LIN {X 0,Y 108.174,Z 556.008,A -85,B 0,C 180,E1 -26292.962,E2 -26292.962} C_VEL
LIN {X 0,Y 107.903,Z 556.034,A -85,B 0,C 180,E1 -26299.008,E2 -26299.008} C_VEL
LIN {X 0,Y 107.859,Z 556.038,A -85,B 0,C 180,E1 -26304.247,E2 -26304.247} C_VEL
LIN {X 0,Y 108.791,Z 558.837,A -85,B 0,C 180,E1 -26305.228,E2 -26305.228} C_VEL
LIN {X 0,Y 110.959,Z 561.09,A -85,B 0,C 180,E1 -26306.828,E2 -26306.828} C_VEL
LIN {X 0,Y 113.315,Z 564.846,A -85,B 0,C 180,E1 -26308.604,E2 -26308.604} C_VEL
LIN {X 0,Y 114.759,Z 566.953,A -85,B 0,C 180,E1 -26309.608,E2 -26309.608} C_VEL
LIN {X 0,Y 119.458,Z 573.968,A -85,B 0,C 180,E1 -26312.627,E2 -26312.627} C_VEL
LIN {X 0,Y 123.093,Z 581.209,A -85,B 0,C 180,E1 -26314.912,E2 -26314.912} C_VEL
LIN {X 0,Y 127.55,Z 591.655,A -85,B 0,C 180,E1 -26317.589,E2 -26317.589} C_VEL
LIN {X 0,Y 132.802,Z 606.179,A -85,B 0,C 180,E1 -26320.632,E2 -26320.632} C_VEL
LIN {X 0,Y 135.067,Z 613.749,A -85,B 0,C 180,E1 -26321.938,E2 -26321.938} C_VEL
LIN {X 0,Y 135.827,Z 626.997,A -85,B 0,C 180,E1 -26323.168,E2 -26323.168} C_VEL
LIN {X 0,Y 132.836,Z 662.155,A -85,B 0,C 180,E1 -26325.068,E2 -26325.068} C_VEL
LIN {X 0,Y 130.992,Z 674.498,A -85,B 0,C 180,E1 -26326.177,E2 -26326.177} C_VEL
LIN {X 0,Y 128.248,Z 687.244,A -85,B 0,C 180,E1 -26327.834,E2 -26327.834} C_VEL
LIN {X 0,Y 124.808,Z 699.792,A -85,B 0,C 180,E1 -26330.17,E2 -26330.17} C_VEL
LIN {X 0,Y 121.198,Z 711.054,A -85,B 0,C 180,E1 -26333.015,E2 -26333.015} C_VEL
LIN {X 0,Y 117.501,Z 721.244,A -85,B 0,C 180,E1 -26336.41,E2 -26336.41} C_VEL
LIN {X 0,Y 113.958,Z 730.437,A -85,B 0,C 180,E1 -26340.438,E2 -26340.438} C_VEL
LIN {X 0,Y 110.529,Z 739.404,A -85,B 0,C 180,E1 -26345.588,E2 -26345.588} C_VEL
LIN {X 0,Y 107.952,Z 746.556,A -85,B 0,C 180,E1 -26351.004,E2 -26351.004} C_VEL
LIN {X 0,Y 106.36,Z 752.228,A -85,B 0,C 180,E1 -26356.628,E2 -26356.628} C_VEL
LIN {X 0,Y 105.688,Z 756.645,A -85,B 0,C 180,E1 -26362.357,E2 -26362.357} C_VEL
LIN {X 0,Y 105.699,Z 758.945,A -85,B 0,C 180,E1 -26366.188,E2 -26366.188} C_VEL
LIN {X 0,Y 105.856,Z 760.773,A -85,B 0,C 180,E1 -26370,E2 -26370} C_VEL
LIN {X 0,Y 105.561,Z 762.058,A -85,B 0,C 180,E1 -26373.817,E2 -26373.817} C_VEL
LIN {X 0,Y 105.804,Z 763.39,A -85,B 0,C 180,E1 -26381.494,E2 -26381.494} C_VEL
LIN {X 0,Y 107.796,Z 763.255,A -85,B 0,C 180,E1 -26389.025,E2 -26389.025} C_VEL
LIN {X 0,Y 111.779,Z 761.601,A -85,B 0,C 180,E1 -26396.111,E2 -26396.111} C_VEL
LIN {X 0,Y 117.427,Z 758.445,A -85,B 0,C 180,E1 -26402.591,E2 -26402.591} C_VEL
LIN {X 0,Y 122.535,Z 755.011,A -85,B 0,C 180,E1 -26407.029,E2 -26407.029} C_VEL
LIN {X 0,Y 128.434,Z 750.585,A -85,B 0,C 180,E1 -26411.043,E2 -26411.043} C_VEL
LIN {X 0,Y 136.128,Z 744.032,A -85,B 0,C 180,E1 -26415.224,E2 -26415.224} C_VEL
LIN {X 0,Y 143.408,Z 736.982,A -85,B 0,C 180,E1 -26418.36,E2 -26418.36} C_VEL
LIN {X 0,Y 151.083,Z 728.338,A -85,B 0,C 180,E1 -26421.183,E2 -26421.183} C_VEL
LIN {X 0,Y 157.807,Z 719.589,A -85,B 0,C 180,E1 -26423.285,E2 -26423.285} C_VEL
LIN {X 0,Y 164.827,Z 708.925,A -85,B 0,C 180,E1 -26425.162,E2 -26425.162} C_VEL
LIN {X 0,Y 166.611,Z 705.818,A -85,B 0,C 180,E1 -26425.606,E2 -26425.606} C_VEL
LIN {X 0,Y 169.05,Z 701.001,A -85,B 0,C 180,E1 -26426.427,E2 -26426.427} C_VEL
LIN {X 0,Y 172.027,Z 693.095,A -85,B 0,C 180,E1 -26428.171,E2 -26428.171} C_VEL
LIN {X 0,Y 174.685,Z 684.872,A -85,B 0,C 180,E1 -26429.755,E2 -26429.755} C_VEL
LIN {X 0,Y 176.474,Z 679.565,A -85,B 0,C 180,E1 -26430.348,E2 -26430.348} C_VEL
LIN {X 0,Y 180.32,Z 666.962,A -85,B 0,C 180,E1 -26431.026,E2 -26431.026} C_VEL
LIN {X 0,Y 183.006,Z 653.633,A -85,B 0,C 180,E1 -26431.546,E2 -26431.546} C_VEL
LIN {X 0,Y 183.302,Z 651.418,A -85,B 0,C 180,E1 -26431.674,E2 -26431.674} C_VEL
LIN {X 0,Y 182.371,Z 646.522,A -85,B 0,C 180,E1 -26434.497,E2 -26434.497} C_VEL
LIN {X 0,Y 181.708,Z 643.146,A -85,B 0,C 180,E1 -26437.408,E2 -26437.408} C_VEL
LIN {X 0,Y 181.435,Z 641.338,A -85,B 0,C 180,E1 -26440.719,E2 -26440.719} C_VEL
LIN {X 0,Y 181.844,Z 641.486,A -85,B 0,C 180,E1 -26445.058,E2 -26445.058} C_VEL
LIN {X 0,Y 182.153,Z 642.109,A -85,B 0,C 180,E1 -26446.471,E2 -26446.471} C_VEL
LIN {X 0,Y 183.563,Z 645.549,A -85,B 0,C 180,E1 -26450.36,E2 -26450.36} C_VEL
LIN {X 0,Y 183.824,Z 646.592,A -85,B 0,C 180,E1 -26451.003,E2 -26451.003} C_VEL
LIN {X 0,Y 181.304,Z 660.599,A -85,B 0,C 180,E1 -26451.676,E2 -26451.676} C_VEL
LIN {X 0,Y 177.981,Z 672.516,A -85,B 0,C 180,E1 -26452.421,E2 -26452.421} C_VEL
LIN {X 0,Y 173.515,Z 684.485,A -85,B 0,C 180,E1 -26453.506,E2 -26453.506} C_VEL
LIN {X 0,Y 167.67,Z 696.546,A -85,B 0,C 180,E1 -26454.962,E2 -26454.962} C_VEL
LIN {X 0,Y 160.872,Z 707.775,A -85,B 0,C 180,E1 -26456.766,E2 -26456.766} C_VEL
LIN {X 0,Y 153.414,Z 717.859,A -85,B 0,C 180,E1 -26459.021,E2 -26459.021} C_VEL
LIN {X 0,Y 146.181,Z 726.118,A -85,B 0,C 180,E1 -26461.47,E2 -26461.47} C_VEL
LIN {X 0,Y 139.25,Z 732.906,A -85,B 0,C 180,E1 -26464.196,E2 -26464.196} C_VEL
LIN {X 0,Y 131.246,Z 739.533,A -85,B 0,C 180,E1 -26467.855,E2 -26467.855} C_VEL
LIN {X 0,Y 125.299,Z 743.757,A -85,B 0,C 180,E1 -26471.127,E2 -26471.127} C_VEL
LIN {X 0,Y 119.48,Z 747.278,A -85,B 0,C 180,E1 -26474.923,E2 -26474.923} C_VEL
LIN {X 0,Y 112.607,Z 750.675,A -85,B 0,C 180,E1 -26480.585,E2 -26480.585} C_VEL
LIN {X 0,Y 106.482,Z 752.713,A -85,B 0,C 180,E1 -26487.515,E2 -26487.515} C_VEL
LIN {X 0,Y 102.231,Z 753.183,A -85,B 0,C 180,E1 -26494.418,E2 -26494.418} C_VEL
LIN {X 0,Y 100.171,Z 752.678,A -85,B 0,C 180,E1 -26499.489,E2 -26499.489} C_VEL
LIN {X 0,Y 98.606,Z 751.336,A -85,B 0,C 180,E1 -26505.455,E2 -26505.455} C_VEL
LIN {X 0,Y 97.956,Z 748.857,A -85,B 0,C 180,E1 -26512.109,E2 -26512.109} C_VEL
LIN {X 0,Y 98.45,Z 745.149,A -85,B 0,C 180,E1 -26518.937,E2 -26518.937} C_VEL
LIN {X 0,Y 100.058,Z 739.9,A -85,B 0,C 180,E1 -26525.934,E2 -26525.934} C_VEL
LIN {X 0,Y 102.102,Z 734.278,A -85,B 0,C 180,E1 -26531.582,E2 -26531.582} C_VEL
LIN {X 0,Y 105.198,Z 726.618,A -85,B 0,C 180,E1 -26537.46,E2 -26537.46} C_VEL
LIN {X 0,Y 108.794,Z 717.855,A -85,B 0,C 180,E1 -26542.577,E2 -26542.577} C_VEL
LIN {X 0,Y 112.615,Z 708.271,A -85,B 0,C 180,E1 -26546.849,E2 -26546.849} C_VEL
LIN {X 0,Y 116.423,Z 697.687,A -85,B 0,C 180,E1 -26550.419,E2 -26550.419} C_VEL
LIN {X 0,Y 120.088,Z 686.177,A -85,B 0,C 180,E1 -26553.355,E2 -26553.355} C_VEL
LIN {X 0,Y 123.278,Z 673.736,A -85,B 0,C 180,E1 -26555.726,E2 -26555.726} C_VEL
LIN {X 0,Y 125.95,Z 660.371,A -85,B 0,C 180,E1 -26557.516,E2 -26557.516} C_VEL
LIN {X 0,Y 127.681,Z 647.584,A -85,B 0,C 180,E1 -26558.677,E2 -26558.677} C_VEL
LIN {X 0,Y 130.987,Z 609.66,A -85,B 0,C 180,E1 -26560.71,E2 -26560.71} C_VEL
LIN {X 0,Y 126.196,Z 597.94,A -85,B 0,C 180,E1 -26563.382,E2 -26563.382} C_VEL
LIN {X 0,Y 118.263,Z 583.132,A -85,B 0,C 180,E1 -26568.048,E2 -26568.048} C_VEL
LIN {X 0,Y 111.781,Z 573.193,A -85,B 0,C 180,E1 -26572.338,E2 -26572.338} C_VEL
LIN {X 0,Y 109.745,Z 570.24,A -85,B 0,C 180,E1 -26573.837,E2 -26573.837} C_VEL
LIN {X 0,Y 107.325,Z 566.668,A -85,B 0,C 180,E1 -26575.766,E2 -26575.766} C_VEL
LIN {X 0,Y 104.957,Z 563.637,A -85,B 0,C 180,E1 -26577.736,E2 -26577.736} C_VEL
LIN {X 0,Y 104.04,Z 562.118,A -85,B 0,C 180,E1 -26578.583,E2 -26578.583} C_VEL
LIN {X 0,Y 101.846,Z 560.004,A -85,B 0,C 180,E1 -26580.508,E2 -26580.508} C_VEL
LIN {X 0,Y 100.884,Z 557.533,A -85,B 0,C 180,E1 -26581.636,E2 -26581.636} C_VEL
LIN {X 0,Y 100.774,Z 556.932,A -85,B 0,C 180,E1 -26581.93,E2 -26581.93} C_VEL
LIN {X 0,Y 100.73,Z 556.92,A -85,B 0,C 180,E1 -26589.875,E2 -26589.875} C_VEL
LIN {X 0,Y 100.746,Z 556.92,A -85,B 0,C 180,E1 -26595.769,E2 -26595.769} C_VEL
LIN {X 0,Y 100.726,Z 556.931,A -85,B 0,C 180,E1 -26601.103,E2 -26601.103} C_VEL
LIN {X 0,Y 100.706,Z 556.915,A -85,B 0,C 180,E1 -26606.869,E2 -26606.869} C_VEL
LIN {X 0,Y 100.783,Z 556.926,A -85,B 0,C 180,E1 -26615.268,E2 -26615.268} C_VEL
LIN {X 0,Y 100.812,Z 556.897,A -85,B 0,C 180,E1 -26619.602,E2 -26619.602} C_VEL
LIN {X 0,Y 101.184,Z 556.859,A -85,B 0,C 180,E1 -26627.975,E2 -26627.975} C_VEL
LIN {X 0,Y 101.263,Z 556.844,A -85,B 0,C 180,E1 -26632.023,E2 -26632.023} C_VEL
LIN {X 0,Y 101.867,Z 556.767,A -85,B 0,C 180,E1 -26640.002,E2 -26640.002} C_VEL
LIN {X 0,Y 101.245,Z 556.856,A -85,B 0,C 180,E1 -26647.982,E2 -26647.982} C_VEL
LIN {X 0,Y 101.103,Z 556.89,A -85,B 0,C 180,E1 -26653.304,E2 -26653.304} C_VEL
LIN {X 0,Y 100.862,Z 557.093,A -85,B 0,C 180,E1 -26659.33,E2 -26659.33} C_VEL
LIN {X 0,Y 101.695,Z 559.548,A -85,B 0,C 180,E1 -26660.349,E2 -26660.349} C_VEL
LIN {X 0,Y 103.691,Z 561.773,A -85,B 0,C 180,E1 -26662.151,E2 -26662.151} C_VEL
LIN {X 0,Y 104.434,Z 562.453,A -85,B 0,C 180,E1 -26662.767,E2 -26662.767} C_VEL
LIN {X 0,Y 106.317,Z 565.65,A -85,B 0,C 180,E1 -26664.46,E2 -26664.46} C_VEL
LIN {X 0,Y 107.94,Z 567.61,A -85,B 0,C 180,E1 -26665.756,E2 -26665.756} C_VEL
LIN {X 0,Y 113.394,Z 575.832,A -85,B 0,C 180,E1 -26669.827,E2 -26669.827} C_VEL
LIN {X 0,Y 116.738,Z 581.563,A -85,B 0,C 180,E1 -26672.094,E2 -26672.094} C_VEL
LIN {X 0,Y 122.043,Z 593.85,A -85,B 0,C 180,E1 -26675.636,E2 -26675.636} C_VEL
LIN {X 0,Y 127.478,Z 609.128,A -85,B 0,C 180,E1 -26679.046,E2 -26679.046} C_VEL
LIN {X 0,Y 129.395,Z 615.319,A -85,B 0,C 180,E1 -26680.23,E2 -26680.23} C_VEL
LIN {X 0,Y 129.944,Z 628.507,A -85,B 0,C 180,E1 -26681.481,E2 -26681.481} C_VEL
LIN {X 0,Y 126.942,Z 661.822,A -85,B 0,C 180,E1 -26683.326,E2 -26683.326} C_VEL
LIN {X 0,Y 124.843,Z 675.074,A -85,B 0,C 180,E1 -26684.564,E2 -26684.564} C_VEL
LIN {X 0,Y 122.013,Z 687.548,A -85,B 0,C 180,E1 -26686.276,E2 -26686.276} C_VEL
LIN {X 0,Y 118.426,Z 699.92,A -85,B 0,C 180,E1 -26688.685,E2 -26688.685} C_VEL
LIN {X 0,Y 114.667,Z 711.088,A -85,B 0,C 180,E1 -26691.644,E2 -26691.644} C_VEL
LIN {X 0,Y 110.828,Z 721.179,A -85,B 0,C 180,E1 -26695.2,E2 -26695.2} C_VEL
LIN {X 0,Y 107.103,Z 730.309,A -85,B 0,C 180,E1 -26699.434,E2 -26699.434} C_VEL
LIN {X 0,Y 103.543,Z 739.234,A -85,B 0,C 180,E1 -26704.899,E2 -26704.899} C_VEL
LIN {X 0,Y 100.866,Z 746.322,A -85,B 0,C 180,E1 -26710.673,E2 -26710.673} C_VEL
LIN {X 0,Y 99.063,Z 752.766,A -85,B 0,C 180,E1 -26717.712,E2 -26717.712} C_VEL
LIN {X 0,Y 98.604,Z 756.946,A -85,B 0,C 180,E1 -26723.863,E2 -26723.863} C_VEL
LIN {X 0,Y 98.792,Z 759.978,A -85,B 0,C 180,E1 -26730,E2 -26730} C_VEL
LIN {X 0,Y 98.48,Z 761.358,A -85,B 0,C 180,E1 -26734.092,E2 -26734.092} C_VEL
LIN {X 0,Y 98.424,Z 762.314,A -85,B 0,C 180,E1 -26738.21,E2 -26738.21} C_VEL
LIN {X 0,Y 99.706,Z 763.05,A -85,B 0,C 180,E1 -26746.376,E2 -26746.376} C_VEL
LIN {X 0,Y 103.03,Z 762.345,A -85,B 0,C 180,E1 -26754.159,E2 -26754.159} C_VEL
LIN {X 0,Y 105.416,Z 761.445,A -85,B 0,C 180,E1 -26757.819,E2 -26757.819} C_VEL
LIN {X 0,Y 111.485,Z 758.462,A -85,B 0,C 180,E1 -26764.565,E2 -26764.565} C_VEL
LIN {X 0,Y 118.928,Z 753.911,A -85,B 0,C 180,E1 -26770.544,E2 -26770.544} C_VEL
LIN {X 0,Y 125.415,Z 749.322,A -85,B 0,C 180,E1 -26774.464,E2 -26774.464} C_VEL
LIN {X 0,Y 133.776,Z 742.537,A -85,B 0,C 180,E1 -26778.47,E2 -26778.47} C_VEL
LIN {X 0,Y 142.731,Z 733.94,A -85,B 0,C 180,E1 -26781.981,E2 -26781.981} C_VEL
LIN {X 0,Y 150.93,Z 724.692,A -85,B 0,C 180,E1 -26784.574,E2 -26784.574} C_VEL
LIN {X 0,Y 158.746,Z 714.242,A -85,B 0,C 180,E1 -26786.68,E2 -26786.68} C_VEL
LIN {X 0,Y 165.375,Z 703.731,A -85,B 0,C 180,E1 -26788.204,E2 -26788.204} C_VEL
LIN {X 0,Y 171.418,Z 691.984,A -85,B 0,C 180,E1 -26789.425,E2 -26789.425} C_VEL
LIN {X 0,Y 176.474,Z 679.565,A -85,B 0,C 180,E1 -26790.348,E2 -26790.348} C_VEL
LIN {X 0,Y 177.566,Z 675.97,A -85,B 0,C 180,E1 -26790.789,E2 -26790.789} C_VEL
LIN {X 0,Y 179.512,Z 664.776,A -85,B 0,C 180,E1 -26793.131,E2 -26793.131} C_VEL
LIN {X 0,Y 180.209,Z 661.025,A -85,B 0,C 180,E1 -26793.496,E2 -26793.496} C_VEL
LIN {X 0,Y 181.288,Z 655.573,A -85,B 0,C 180,E1 -26793.701,E2 -26793.701} C_VEL
LIN {X 0,Y 180.849,Z 652.395,A -85,B 0,C 180,E1 -26795.779,E2 -26795.779} C_VEL
LIN {X 0,Y 180.526,Z 649.844,A -85,B 0,C 180,E1 -26798.12,E2 -26798.12} C_VEL
LIN {X 0,Y 180.385,Z 648.406,A -85,B 0,C 180,E1 -26800.602,E2 -26800.602} C_VEL
LIN {X 0,Y 180.635,Z 648.307,A -85,B 0,C 180,E1 -26804.195,E2 -26804.195} C_VEL
LIN {X 0,Y 180.93,Z 648.948,A -85,B 0,C 180,E1 -26805.948,E2 -26805.948} C_VEL
LIN {X 0,Y 181.783,Z 651.483,A -85,B 0,C 180,E1 -26808.985,E2 -26808.985} C_VEL
LIN {X 0,Y 178.929,Z 664.632,A -85,B 0,C 180,E1 -26809.663,E2 -26809.663} C_VEL
LIN {X 0,Y 175.422,Z 675.737,A -85,B 0,C 180,E1 -26810.391,E2 -26810.391} C_VEL
LIN {X 0,Y 170.55,Z 687.561,A -85,B 0,C 180,E1 -26811.481,E2 -26811.481} C_VEL
LIN {X 0,Y 164.386,Z 699.333,A -85,B 0,C 180,E1 -26812.918,E2 -26812.918} C_VEL
LIN {X 0,Y 157.501,Z 709.886,A -85,B 0,C 180,E1 -26814.627,E2 -26814.627} C_VEL
LIN {X 0,Y 149.558,Z 719.987,A -85,B 0,C 180,E1 -26816.888,E2 -26816.888} C_VEL
LIN {X 0,Y 142.328,Z 727.638,A -85,B 0,C 180,E1 -26819.191,E2 -26819.191} C_VEL
LIN {X 0,Y 133.649,Z 735.359,A -85,B 0,C 180,E1 -26822.428,E2 -26822.428} C_VEL
LIN {X 0,Y 124.692,Z 742.032,A -85,B 0,C 180,E1 -26826.471,E2 -26826.471} C_VEL
LIN {X 0,Y 117.771,Z 746.289,A -85,B 0,C 180,E1 -26830.311,E2 -26830.311} C_VEL
LIN {X 0,Y 109.665,Z 750.263,A -85,B 0,C 180,E1 -26836,E2 -26836} C_VEL
LIN {X 0,Y 104.893,Z 752.074,A -85,B 0,C 180,E1 -26840.282,E2 -26840.282} C_VEL
LIN {X 0,Y 100.767,Z 753.166,A -85,B 0,C 180,E1 -26844.952,E2 -26844.952} C_VEL
LIN {X 0,Y 96.946,Z 753.621,A -85,B 0,C 180,E1 -26850.492,E2 -26850.492} C_VEL
LIN {X 0,Y 93.915,Z 753.228,A -85,B 0,C 180,E1 -26856.772,E2 -26856.772} C_VEL
LIN {X 0,Y 91.867,Z 751.887,A -85,B 0,C 180,E1 -26863.51,E2 -26863.51} C_VEL
LIN {X 0,Y 90.882,Z 748.999,A -85,B 0,C 180,E1 -26871.784,E2 -26871.784} C_VEL
LIN {X 0,Y 91.592,Z 744.432,A -85,B 0,C 180,E1 -26880.37,E2 -26880.37} C_VEL
LIN {X 0,Y 93.465,Z 738.703,A -85,B 0,C 180,E1 -26887.916,E2 -26887.916} C_VEL
LIN {X 0,Y 95.974,Z 732.381,A -85,B 0,C 180,E1 -26894.178,E2 -26894.178} C_VEL
LIN {X 0,Y 99.392,Z 724.525,A -85,B 0,C 180,E1 -26900.101,E2 -26900.101} C_VEL
LIN {X 0,Y 103.613,Z 714.664,A -85,B 0,C 180,E1 -26905.624,E2 -26905.624} C_VEL
LIN {X 0,Y 107.806,Z 704.231,A -85,B 0,C 180,E1 -26910,E2 -26910} C_VEL
LIN {X 0,Y 111.982,Z 692.588,A -85,B 0,C 180,E1 -26913.598,E2 -26913.598} C_VEL
LIN {X 0,Y 115.588,Z 680.766,A -85,B 0,C 180,E1 -26916.327,E2 -26916.327} C_VEL
LIN {X 0,Y 118.473,Z 669.013,A -85,B 0,C 180,E1 -26918.314,E2 -26918.314} C_VEL
LIN {X 0,Y 120.883,Z 655.475,A -85,B 0,C 180,E1 -26919.939,E2 -26919.939} C_VEL
LIN {X 0,Y 122.474,Z 642.382,A -85,B 0,C 180,E1 -26920.909,E2 -26920.909} C_VEL
LIN {X 0,Y 125.157,Z 611.497,A -85,B 0,C 180,E1 -26922.599,E2 -26922.599} C_VEL
LIN {X 0,Y 121.457,Z 602.23,A -85,B 0,C 180,E1 -26924.84,E2 -26924.84} C_VEL
LIN {X 0,Y 114.318,Z 588.414,A -85,B 0,C 180,E1 -26929.398,E2 -26929.398} C_VEL
LIN {X 0,Y 108.146,Z 578.586,A -85,B 0,C 180,E1 -26933.816,E2 -26933.816} C_VEL
LIN {X 0,Y 103.85,Z 572.191,A -85,B 0,C 180,E1 -26937.391,E2 -26937.391} C_VEL
LIN {X 0,Y 101.308,Z 568.556,A -85,B 0,C 180,E1 -26939.715,E2 -26939.715} C_VEL
LIN {X 0,Y 98.51,Z 565.258,A -85,B 0,C 180,E1 -26942.472,E2 -26942.472} C_VEL
LIN {X 0,Y 97.581,Z 563.315,A -85,B 0,C 180,E1 -26943.605,E2 -26943.605} C_VEL
LIN {X 0,Y 95.114,Z 561.387,A -85,B 0,C 180,E1 -26946.289,E2 -26946.289} C_VEL
LIN {X 0,Y 93.877,Z 558.999,A -85,B 0,C 180,E1 -26948.013,E2 -26948.013} C_VEL
LIN {X 0,Y 93.661,Z 557.799,A -85,B 0,C 180,E1 -26948.667,E2 -26948.667} C_VEL
LIN {X 0,Y 93.646,Z 557.818,A -85,B 0,C 180,E1 -26952.487,E2 -26952.487} C_VEL
LIN {X 0,Y 93.643,Z 557.795,A -85,B 0,C 180,E1 -26958.633,E2 -26958.633} C_VEL
LIN {X 0,Y 93.62,Z 557.804,A -85,B 0,C 180,E1 -26965.664,E2 -26965.664} C_VEL
LIN {X 0,Y 93.666,Z 557.817,A -85,B 0,C 180,E1 -26974.207,E2 -26974.207} C_VEL
LIN {X 0,Y 93.688,Z 557.786,A -85,B 0,C 180,E1 -26977.973,E2 -26977.973} C_VEL
LIN {X 0,Y 94.088,Z 557.751,A -85,B 0,C 180,E1 -26987.053,E2 -26987.053} C_VEL
LIN {X 0,Y 94.196,Z 557.72,A -85,B 0,C 180,E1 -26991.42,E2 -26991.42} C_VEL
LIN {X 0,Y 94.793,Z 557.647,A -85,B 0,C 180,E1 -27000.002,E2 -27000.002} C_VEL
LIN {X 0,Y 94.177,Z 557.733,A -85,B 0,C 180,E1 -27008.586,E2 -27008.586} C_VEL
LIN {X 0,Y 94.077,Z 557.764,A -85,B 0,C 180,E1 -27012.953,E2 -27012.953} C_VEL
LIN {X 0,Y 94.789,Z 560.311,A -85,B 0,C 180,E1 -27014.208,E2 -27014.208} C_VEL
LIN {X 0,Y 96.581,Z 562.529,A -85,B 0,C 180,E1 -27016.387,E2 -27016.387} C_VEL
LIN {X 0,Y 97.783,Z 563.493,A -85,B 0,C 180,E1 -27017.653,E2 -27017.653} C_VEL
LIN {X 0,Y 99.624,Z 566.67,A -85,B 0,C 180,E1 -27019.714,E2 -27019.714} C_VEL
LIN {X 0,Y 101.343,Z 568.577,A -85,B 0,C 180,E1 -27021.339,E2 -27021.339} C_VEL
LIN {X 0,Y 103.777,Z 572.135,A -85,B 0,C 180,E1 -27023.564,E2 -27023.564} C_VEL
LIN {X 0,Y 109.381,Z 580.683,A -85,B 0,C 180,E1 -27028.157,E2 -27028.157} C_VEL
LIN {X 0,Y 112.465,Z 586.164,A -85,B 0,C 180,E1 -27030.434,E2 -27030.434} C_VEL
LIN {X 0,Y 117.395,Z 598.14,A -85,B 0,C 180,E1 -27034.047,E2 -27034.047} C_VEL
LIN {X 0,Y 122.249,Z 612.383,A -85,B 0,C 180,E1 -27037.391,E2 -27037.391} C_VEL
LIN {X 0,Y 123.866,Z 618.008,A -85,B 0,C 180,E1 -27038.49,E2 -27038.49} C_VEL
LIN {X 0,Y 124.205,Z 629.468,A -85,B 0,C 180,E1 -27039.601,E2 -27039.601} C_VEL
LIN {X 0,Y 121.204,Z 661.249,A -85,B 0,C 180,E1 -27041.395,E2 -27041.395} C_VEL
LIN {X 0,Y 119.119,Z 674.228,A -85,B 0,C 180,E1 -27042.639,E2 -27042.639} C_VEL
LIN {X 0,Y 116.147,Z 686.797,A -85,B 0,C 180,E1 -27044.377,E2 -27044.377} C_VEL
LIN {X 0,Y 112.659,Z 698.443,A -85,B 0,C 180,E1 -27046.67,E2 -27046.67} C_VEL
LIN {X 0,Y 108.7,Z 709.784,A -85,B 0,C 180,E1 -27049.719,E2 -27049.719} C_VEL
LIN {X 0,Y 105.062,Z 718.997,A -85,B 0,C 180,E1 -27052.985,E2 -27052.985} C_VEL
LIN {X 0,Y 101.042,Z 728.481,A -85,B 0,C 180,E1 -27057.382,E2 -27057.382} C_VEL
LIN {X 0,Y 97.114,Z 737.62,A -85,B 0,C 180,E1 -27063.109,E2 -27063.109} C_VEL
LIN {X 0,Y 94.187,Z 744.963,A -85,B 0,C 180,E1 -27069.242,E2 -27069.242} C_VEL
LIN {X 0,Y 92.548,Z 749.899,A -85,B 0,C 180,E1 -27074.587,E2 -27074.587} C_VEL
LIN {X 0,Y 91.622,Z 754.658,A -85,B 0,C 180,E1 -27081.175,E2 -27081.175} C_VEL
LIN {X 0,Y 91.588,Z 757.393,A -85,B 0,C 180,E1 -27086.024,E2 -27086.024} C_VEL
LIN {X 0,Y 91.73,Z 759.166,A -85,B 0,C 180,E1 -27090,E2 -27090} C_VEL
LIN {X 0,Y 91.411,Z 760.618,A -85,B 0,C 180,E1 -27094.409,E2 -27094.409} C_VEL
LIN {X 0,Y 91.9,Z 762.332,A -85,B 0,C 180,E1 -27103.263,E2 -27103.263} C_VEL
LIN {X 0,Y 94.422,Z 762.497,A -85,B 0,C 180,E1 -27111.848,E2 -27111.848} C_VEL
LIN {X 0,Y 99.161,Z 761.233,A -85,B 0,C 180,E1 -27119.743,E2 -27119.743} C_VEL
LIN {X 0,Y 105.693,Z 758.48,A -85,B 0,C 180,E1 -27126.758,E2 -27126.758} C_VEL
LIN {X 0,Y 113.615,Z 754.137,A -85,B 0,C 180,E1 -27132.876,E2 -27132.876} C_VEL
LIN {X 0,Y 120.47,Z 749.748,A -85,B 0,C 180,E1 -27136.82,E2 -27136.82} C_VEL
LIN {X 0,Y 129.201,Z 743.244,A -85,B 0,C 180,E1 -27140.816,E2 -27140.816} C_VEL
LIN {X 0,Y 138.515,Z 734.952,A -85,B 0,C 180,E1 -27144.271,E2 -27144.271} C_VEL
LIN {X 0,Y 146.99,Z 726.121,A -85,B 0,C 180,E1 -27146.793,E2 -27146.793} C_VEL
LIN {X 0,Y 155.052,Z 716.15,A -85,B 0,C 180,E1 -27148.817,E2 -27148.817} C_VEL
LIN {X 0,Y 162.581,Z 704.863,A -85,B 0,C 180,E1 -27150.451,E2 -27150.451} C_VEL
LIN {X 0,Y 168.768,Z 693.602,A -85,B 0,C 180,E1 -27151.604,E2 -27151.604} C_VEL
LIN {X 0,Y 174.518,Z 680.239,A -85,B 0,C 180,E1 -27152.562,E2 -27152.562} C_VEL
LIN {X 0,Y 178.785,Z 666.964,A -85,B 0,C 180,E1 -27153.238,E2 -27153.238} C_VEL
LIN {X 0,Y 180.209,Z 661.025,A -85,B 0,C 180,E1 -27153.496,E2 -27153.496} C_VEL
LIN {X 0,Y 180.487,Z 659.028,A -85,B 0,C 180,E1 -27153.833,E2 -27153.833} C_VEL
LIN {X 0,Y 180.462,Z 657.363,A -85,B 0,C 180,E1 -27154.636,E2 -27154.636} C_VEL
LIN {X 0,Y 180.075,Z 656.344,A -85,B 0,C 180,E1 -27156.041,E2 -27156.041} C_VEL
LIN {X 0,Y 179.126,Z 656.066,A -85,B 0,C 180,E1 -27159.577,E2 -27159.577} C_VEL
LIN {X 0,Y 179.108,Z 655.824,A -85,B 0,C 180,E1 -27160.078,E2 -27160.078} C_VEL
LIN {X 0,Y 179.118,Z 655.203,A -85,B 0,C 180,E1 -27161.705,E2 -27161.705} C_VEL
LIN {X 0,Y 179.507,Z 655.551,A -85,B 0,C 180,E1 -27165.248,E2 -27165.248} C_VEL
LIN {X 0,Y 179.709,Z 657.068,A -85,B 0,C 180,E1 -27167.008,E2 -27167.008} C_VEL
LIN {X 0,Y 176.409,Z 669.66,A -85,B 0,C 180,E1 -27167.655,E2 -27167.655} C_VEL
LIN {X 0,Y 171.611,Z 682.589,A -85,B 0,C 180,E1 -27168.606,E2 -27168.606} C_VEL
LIN {X 0,Y 166.028,Z 694.169,A -85,B 0,C 180,E1 -27169.779,E2 -27169.779} C_VEL
LIN {X 0,Y 159.079,Z 705.518,A -85,B 0,C 180,E1 -27171.298,E2 -27171.298} C_VEL
LIN {X 0,Y 152.252,Z 714.701,A -85,B 0,C 180,E1 -27172.941,E2 -27172.941} C_VEL
LIN {X 0,Y 144.482,Z 723.512,A -85,B 0,C 180,E1 -27175.043,E2 -27175.043} C_VEL
LIN {X 0,Y 135.679,Z 731.834,A -85,B 0,C 180,E1 -27177.779,E2 -27177.779} C_VEL
LIN {X 0,Y 126.528,Z 738.973,A -85,B 0,C 180,E1 -27181.189,E2 -27181.189} C_VEL
LIN {X 0,Y 119.787,Z 743.385,A -85,B 0,C 180,E1 -27184.15,E2 -27184.15} C_VEL
LIN {X 0,Y 110.388,Z 748.485,A -85,B 0,C 180,E1 -27189.318,E2 -27189.318} C_VEL
LIN {X 0,Y 102.041,Z 751.849,A -85,B 0,C 180,E1 -27195.374,E2 -27195.374} C_VEL
LIN {X 0,Y 95.78,Z 753.534,A -85,B 0,C 180,E1 -27201.521,E2 -27201.521} C_VEL
LIN {X 0,Y 91.209,Z 754.067,A -85,B 0,C 180,E1 -27207.534,E2 -27207.534} C_VEL
LIN {X 0,Y 86.898,Z 753.457,A -85,B 0,C 180,E1 -27216.027,E2 -27216.027} C_VEL
LIN {X 0,Y 85.054,Z 752.247,A -85,B 0,C 180,E1 -27221.957,E2 -27221.957} C_VEL
LIN {X 0,Y 83.805,Z 749.078,A -85,B 0,C 180,E1 -27231.492,E2 -27231.492} C_VEL
LIN {X 0,Y 84.38,Z 744.813,A -85,B 0,C 180,E1 -27240.018,E2 -27240.018} C_VEL
LIN {X 0,Y 86.434,Z 738.813,A -85,B 0,C 180,E1 -27248.538,E2 -27248.538} C_VEL
LIN {X 0,Y 88.866,Z 732.977,A -85,B 0,C 180,E1 -27254.759,E2 -27254.759} C_VEL
LIN {X 0,Y 92.543,Z 724.951,A -85,B 0,C 180,E1 -27261.264,E2 -27261.264} C_VEL
LIN {X 0,Y 96.545,Z 716.087,A -85,B 0,C 180,E1 -27266.605,E2 -27266.605} C_VEL
LIN {X 0,Y 101.195,Z 705.215,A -85,B 0,C 180,E1 -27271.492,E2 -27271.492} C_VEL
LIN {X 0,Y 105.07,Z 695.19,A -85,B 0,C 180,E1 -27274.838,E2 -27274.838} C_VEL
LIN {X 0,Y 109.058,Z 683.033,A -85,B 0,C 180,E1 -27277.871,E2 -27277.871} C_VEL
LIN {X 0,Y 112.344,Z 670.656,A -85,B 0,C 180,E1 -27280.133,E2 -27280.133} C_VEL
LIN {X 0,Y 114.861,Z 657.82,A -85,B 0,C 180,E1 -27281.775,E2 -27281.775} C_VEL
LIN {X 0,Y 116.717,Z 644.153,A -85,B 0,C 180,E1 -27282.87,E2 -27282.87} C_VEL
LIN {X 0,Y 119.53,Z 614.275,A -85,B 0,C 180,E1 -27284.515,E2 -27284.515} C_VEL
LIN {X 0,Y 119.018,Z 612.229,A -85,B 0,C 180,E1 -27284.916,E2 -27284.916} C_VEL
LIN {X 0,Y 116.634,Z 606.127,A -85,B 0,C 180,E1 -27286.53,E2 -27286.53} C_VEL
LIN {X 0,Y 109.897,Z 592.771,A -85,B 0,C 180,E1 -27291.199,E2 -27291.199} C_VEL
LIN {X 0,Y 103.336,Z 581.898,A -85,B 0,C 180,E1 -27296.487,E2 -27296.487} C_VEL
LIN {X 0,Y 99.931,Z 577.057,A -85,B 0,C 180,E1 -27299.569,E2 -27299.569} C_VEL
LIN {X 0,Y 97.593,Z 573.734,A -85,B 0,C 180,E1 -27301.957,E2 -27301.957} C_VEL
LIN {X 0,Y 95.178,Z 570.274,A -85,B 0,C 180,E1 -27304.714,E2 -27304.714} C_VEL
LIN {X 0,Y 94.58,Z 569.401,A -85,B 0,C 180,E1 -27305.444,E2 -27305.444} C_VEL
LIN {X 0,Y 92.116,Z 566.856,A -85,B 0,C 180,E1 -27308.481,E2 -27308.481} C_VEL
LIN {X 0,Y 90.825,Z 564.314,A -85,B 0,C 180,E1 -27310.506,E2 -27310.506} C_VEL
LIN {X 0,Y 88.01,Z 562.227,A -85,B 0,C 180,E1 -27314.851,E2 -27314.851} C_VEL
LIN {X 0,Y 86.896,Z 560.043,A -85,B 0,C 180,E1 -27317.216,E2 -27317.216} C_VEL
LIN {X 0,Y 86.602,Z 558.671,A -85,B 0,C 180,E1 -27318.16,E2 -27318.16} C_VEL
LIN {X 0,Y 86.57,Z 558.683,A -85,B 0,C 180,E1 -27325.373,E2 -27325.373} C_VEL
LIN {X 0,Y 86.581,Z 558.7,A -85,B 0,C 180,E1 -27333.237,E2 -27333.237} C_VEL
LIN {X 0,Y 86.642,Z 558.665,A -85,B 0,C 180,E1 -27341.07,E2 -27341.07} C_VEL
LIN {X 0,Y 86.967,Z 558.646,A -85,B 0,C 180,E1 -27345.972,E2 -27345.972} C_VEL
LIN {X 0,Y 87.104,Z 558.601,A -85,B 0,C 180,E1 -27350.716,E2 -27350.716} C_VEL
LIN {X 0,Y 87.721,Z 558.528,A -85,B 0,C 180,E1 -27360.002,E2 -27360.002} C_VEL
LIN {X 0,Y 87.271,Z 558.605,A -85,B 0,C 180,E1 -27364.043,E2 -27364.043} C_VEL
LIN {X 0,Y 87.865,Z 560.92,A -85,B 0,C 180,E1 -27365.597,E2 -27365.597} C_VEL
LIN {X 0,Y 89.645,Z 563.215,A -85,B 0,C 180,E1 -27368.739,E2 -27368.739} C_VEL
LIN {X 0,Y 91.398,Z 564.504,A -85,B 0,C 180,E1 -27371.226,E2 -27371.226} C_VEL
LIN {X 0,Y 93.01,Z 567.586,A -85,B 0,C 180,E1 -27373.621,E2 -27373.621} C_VEL
LIN {X 0,Y 95.062,Z 569.835,A -85,B 0,C 180,E1 -27376.141,E2 -27376.141} C_VEL
LIN {X 0,Y 97.508,Z 573.495,A -85,B 0,C 180,E1 -27378.962,E2 -27378.962} C_VEL
LIN {X 0,Y 98.888,Z 575.542,A -85,B 0,C 180,E1 -27380.409,E2 -27380.409} C_VEL
LIN {X 0,Y 101.918,Z 580.045,A -85,B 0,C 180,E1 -27383.304,E2 -27383.304} C_VEL
LIN {X 0,Y 105.825,Z 586.251,A -85,B 0,C 180,E1 -27386.695,E2 -27386.695} C_VEL
LIN {X 0,Y 108.188,Z 590.603,A -85,B 0,C 180,E1 -27388.611,E2 -27388.611} C_VEL
LIN {X 0,Y 112.866,Z 602.453,A -85,B 0,C 180,E1 -27392.344,E2 -27392.344} C_VEL
LIN {X 0,Y 117.303,Z 616.175,A -85,B 0,C 180,E1 -27395.745,E2 -27395.745} C_VEL
LIN {X 0,Y 118.368,Z 620.399,A -85,B 0,C 180,E1 -27396.586,E2 -27396.586} C_VEL
LIN {X 0,Y 118.642,Z 629.302,A -85,B 0,C 180,E1 -27397.518,E2 -27397.518} C_VEL
LIN {X 0,Y 115.562,Z 660.655,A -85,B 0,C 180,E1 -27399.332,E2 -27399.332} C_VEL
LIN {X 0,Y 113.378,Z 673.671,A -85,B 0,C 180,E1 -27400.595,E2 -27400.595} C_VEL
LIN {X 0,Y 110.146,Z 686.792,A -85,B 0,C 180,E1 -27402.461,E2 -27402.461} C_VEL
LIN {X 0,Y 106.511,Z 698.349,A -85,B 0,C 180,E1 -27404.821,E2 -27404.821} C_VEL
LIN {X 0,Y 102.371,Z 709.635,A -85,B 0,C 180,E1 -27407.983,E2 -27407.983} C_VEL
LIN {X 0,Y 98.45,Z 719.038,A -85,B 0,C 180,E1 -27411.49,E2 -27411.49} C_VEL
LIN {X 0,Y 94.32,Z 728.236,A -85,B 0,C 180,E1 -27416.025,E2 -27416.025} C_VEL
LIN {X 0,Y 90.205,Z 737.35,A -85,B 0,C 180,E1 -27422.131,E2 -27422.131} C_VEL
LIN {X 0,Y 87.121,Z 744.662,A -85,B 0,C 180,E1 -27428.715,E2 -27428.715} C_VEL
LIN {X 0,Y 85.196,Z 750.473,A -85,B 0,C 180,E1 -27435.672,E2 -27435.672} C_VEL
LIN {X 0,Y 84.484,Z 754.998,A -85,B 0,C 180,E1 -27442.832,E2 -27442.832} C_VEL
LIN {X 0,Y 84.67,Z 758.353,A -85,B 0,C 180,E1 -27450,E2 -27450} C_VEL
LIN {X 0,Y 84.345,Z 759.869,A -85,B 0,C 180,E1 -27454.78,E2 -27454.78} C_VEL
LIN {X 0,Y 85.001,Z 761.725,A -85,B 0,C 180,E1 -27464.361,E2 -27464.361} C_VEL
LIN {X 0,Y 87.841,Z 762.116,A -85,B 0,C 180,E1 -27473.58,E2 -27473.58} C_VEL
LIN {X 0,Y 93.035,Z 761.016,A -85,B 0,C 180,E1 -27481.923,E2 -27481.923} C_VEL
LIN {X 0,Y 100.079,Z 758.481,A -85,B 0,C 180,E1 -27489.198,E2 -27489.198} C_VEL
LIN {X 0,Y 106.274,Z 755.547,A -85,B 0,C 180,E1 -27493.976,E2 -27493.976} C_VEL
LIN {X 0,Y 113.253,Z 751.675,A -85,B 0,C 180,E1 -27498.129,E2 -27498.129} C_VEL
LIN {X 0,Y 120.843,Z 746.796,A -85,B 0,C 180,E1 -27501.731,E2 -27501.731} C_VEL
LIN {X 0,Y 130.356,Z 739.643,A -85,B 0,C 180,E1 -27505.303,E2 -27505.303} C_VEL
LIN {X 0,Y 138.878,Z 731.989,A -85,B 0,C 180,E1 -27507.954,E2 -27507.954} C_VEL
LIN {X 0,Y 147.764,Z 722.517,A -85,B 0,C 180,E1 -27510.226,E2 -27510.226} C_VEL
LIN {X 0,Y 156.166,Z 711.856,A -85,B 0,C 180,E1 -27512.027,E2 -27512.027} C_VEL
LIN {X 0,Y 163.205,Z 700.971,A -85,B 0,C 180,E1 -27513.319,E2 -27513.319} C_VEL
LIN {X 0,Y 169.587,Z 688.812,A -85,B 0,C 180,E1 -27514.335,E2 -27514.335} C_VEL
LIN {X 0,Y 174.205,Z 677.667,A -85,B 0,C 180,E1 -27515.001,E2 -27515.001} C_VEL
LIN {X 0,Y 178.265,Z 664.418,A -85,B 0,C 180,E1 -27515.607,E2 -27515.607} C_VEL
LIN {X 0,Y 179.314,Z 660.071,A -85,B 0,C 180,E1 -27515.756,E2 -27515.756} C_VEL
LIN {X 0,Y 179.185,Z 657.061,A -85,B 0,C 180,E1 -27518.1,E2 -27518.1} C_VEL
LIN {X 0,Y 179.108,Z 655.824,A -85,B 0,C 180,E1 -27520.078,E2 -27520.078} C_VEL
LIN {X 0,Y 179.02,Z 655.898,A -85,B 0,C 180,E1 -27521.19,E2 -27521.19} C_VEL
LIN {X 0,Y 178.715,Z 657.427,A -85,B 0,C 180,E1 -27522.457,E2 -27522.457} C_VEL
LIN {X 0,Y 178.096,Z 660.501,A -85,B 0,C 180,E1 -27523.738,E2 -27523.738} C_VEL
LIN {X 0,Y 177.334,Z 663.92,A -85,B 0,C 180,E1 -27524.632,E2 -27524.632} C_VEL
LIN {X 0,Y 176.267,Z 667.818,A -85,B 0,C 180,E1 -27525.217,E2 -27525.217} C_VEL
LIN {X 0,Y 175.856,Z 669.2,A -85,B 0,C 180,E1 -27525.324,E2 -27525.324} C_VEL
LIN {X 0,Y 171.401,Z 681.244,A -85,B 0,C 180,E1 -27526.119,E2 -27526.119} C_VEL
LIN {X 0,Y 165.789,Z 692.864,A -85,B 0,C 180,E1 -27527.155,E2 -27527.155} C_VEL
LIN {X 0,Y 159.438,Z 703.469,A -85,B 0,C 180,E1 -27528.408,E2 -27528.408} C_VEL
LIN {X 0,Y 152.663,Z 712.769,A -85,B 0,C 180,E1 -27529.822,E2 -27529.822} C_VEL
LIN {X 0,Y 144.082,Z 722.48,A -85,B 0,C 180,E1 -27531.875,E2 -27531.875} C_VEL
LIN {X 0,Y 135.977,Z 730.117,A -85,B 0,C 180,E1 -27534.065,E2 -27534.065} C_VEL
LIN {X 0,Y 126.668,Z 737.473,A -85,B 0,C 180,E1 -27537.055,E2 -27537.055} C_VEL
LIN {X 0,Y 118.939,Z 742.559,A -85,B 0,C 180,E1 -27539.998,E2 -27539.998} C_VEL
LIN {X 0,Y 111.006,Z 746.918,A -85,B 0,C 180,E1 -27543.628,E2 -27543.628} C_VEL
LIN {X 0,Y 103.612,Z 750.208,A -85,B 0,C 180,E1 -27547.795,E2 -27547.795} C_VEL
LIN {X 0,Y 96.856,Z 752.529,A -85,B 0,C 180,E1 -27552.571,E2 -27552.571} C_VEL
LIN {X 0,Y 89.482,Z 754.206,A -85,B 0,C 180,E1 -27559.53,E2 -27559.53} C_VEL
LIN {X 0,Y 85.243,Z 754.52,A -85,B 0,C 180,E1 -27564.921,E2 -27564.921} C_VEL
LIN {X 0,Y 81.683,Z 754.196,A -85,B 0,C 180,E1 -27571.077,E2 -27571.077} C_VEL
LIN {X 0,Y 78.688,Z 752.949,A -85,B 0,C 180,E1 -27578.694,E2 -27578.694} C_VEL
LIN {X 0,Y 77.023,Z 750.694,A -85,B 0,C 180,E1 -27586.88,E2 -27586.88} C_VEL
LIN {X 0,Y 76.892,Z 746.636,A -85,B 0,C 180,E1 -27596.743,E2 -27596.743} C_VEL
LIN {X 0,Y 78.037,Z 742.424,A -85,B 0,C 180,E1 -27604.231,E2 -27604.231} C_VEL
LIN {X 0,Y 80.126,Z 737.165,A -85,B 0,C 180,E1 -27611.39,E2 -27611.39} C_VEL
LIN {X 0,Y 83.583,Z 729.638,A -85,B 0,C 180,E1 -27619.095,E2 -27619.095} C_VEL
LIN {X 0,Y 87.628,Z 721.28,A -85,B 0,C 180,E1 -27625.4,E2 -27625.4} C_VEL
LIN {X 0,Y 92.012,Z 712.053,A -85,B 0,C 180,E1 -27630.547,E2 -27630.547} C_VEL
LIN {X 0,Y 96.652,Z 701.36,A -85,B 0,C 180,E1 -27634.998,E2 -27634.998} C_VEL
LIN {X 0,Y 101.047,Z 689.818,A -85,B 0,C 180,E1 -27638.499,E2 -27638.499} C_VEL
LIN {X 0,Y 105.095,Z 676.943,A -85,B 0,C 180,E1 -27641.328,E2 -27641.328} C_VEL
LIN {X 0,Y 108.184,Z 664.23,A -85,B 0,C 180,E1 -27643.295,E2 -27643.295} C_VEL
LIN {X 0,Y 110.5,Z 650.388,A -85,B 0,C 180,E1 -27644.738,E2 -27644.738} C_VEL
LIN {X 0,Y 114.014,Z 615.508,A -85,B 0,C 180,E1 -27646.794,E2 -27646.794} C_VEL
LIN {X 0,Y 111.943,Z 610.191,A -85,B 0,C 180,E1 -27648.295,E2 -27648.295} C_VEL
LIN {X 0,Y 105.791,Z 597.449,A -85,B 0,C 180,E1 -27652.991,E2 -27652.991} C_VEL
LIN {X 0,Y 99.63,Z 587.006,A -85,B 0,C 180,E1 -27658.403,E2 -27658.403} C_VEL
LIN {X 0,Y 94.931,Z 579.885,A -85,B 0,C 180,E1 -27663.359,E2 -27663.359} C_VEL
LIN {X 0,Y 92.363,Z 576.135,A -85,B 0,C 180,E1 -27666.504,E2 -27666.504} C_VEL
LIN {X 0,Y 89.398,Z 572.52,A -85,B 0,C 180,E1 -27670.585,E2 -27670.585} C_VEL
LIN {X 0,Y 88.452,Z 570.75,A -85,B 0,C 180,E1 -27672.216,E2 -27672.216} C_VEL
LIN {X 0,Y 86.014,Z 568.593,A -85,B 0,C 180,E1 -27676.416,E2 -27676.416} C_VEL
LIN {X 0,Y 84.688,Z 565.79,A -85,B 0,C 180,E1 -27679.587,E2 -27679.587} C_VEL
LIN {X 0,Y 84.004,Z 565.334,A -85,B 0,C 180,E1 -27681.14,E2 -27681.14} C_VEL
LIN {X 0,Y 80.349,Z 562.115,A -85,B 0,C 180,E1 -27696.823,E2 -27696.823} C_VEL
LIN {X 0,Y 80.605,Z 561.809,A -85,B 0,C 180,E1 -27706.313,E2 -27706.313} C_VEL
LIN {X 0,Y 85.15,Z 565.301,A -85,B 0,C 180,E1 -27722.131,E2 -27722.131} C_VEL
LIN {X 0,Y 86.386,Z 568.248,A -85,B 0,C 180,E1 -27725.107,E2 -27725.107} C_VEL
LIN {X 0,Y 89.053,Z 571.015,A -85,B 0,C 180,E1 -27729.657,E2 -27729.657} C_VEL
LIN {X 0,Y 91.009,Z 574.334,A -85,B 0,C 180,E1 -27732.688,E2 -27732.688} C_VEL
LIN {X 0,Y 92.466,Z 576.093,A -85,B 0,C 180,E1 -27734.585,E2 -27734.585} C_VEL
LIN {X 0,Y 95.821,Z 581.277,A -85,B 0,C 180,E1 -27738.701,E2 -27738.701} C_VEL
LIN {X 0,Y 99.795,Z 587.428,A -85,B 0,C 180,E1 -27742.771,E2 -27742.771} C_VEL
LIN {X 0,Y 103.962,Z 594.937,A -85,B 0,C 180,E1 -27746.591,E2 -27746.591} C_VEL
LIN {X 0,Y 108.158,Z 606.108,A -85,B 0,C 180,E1 -27750.345,E2 -27750.345} C_VEL
LIN {X 0,Y 112.541,Z 620.27,A -85,B 0,C 180,E1 -27754.029,E2 -27754.029} C_VEL
LIN {X 0,Y 113.064,Z 622.764,A -85,B 0,C 180,E1 -27754.524,E2 -27754.524} C_VEL
LIN {X 0,Y 113.089,Z 630.842,A -85,B 0,C 180,E1 -27755.345,E2 -27755.345} C_VEL
LIN {X 0,Y 109.934,Z 660.976,A -85,B 0,C 180,E1 -27757.13,E2 -27757.13} C_VEL
LIN {X 0,Y 107.643,Z 673.831,A -85,B 0,C 180,E1 -27758.421,E2 -27758.421} C_VEL
LIN {X 0,Y 104.552,Z 685.747,A -85,B 0,C 180,E1 -27760.128,E2 -27760.128} C_VEL
LIN {X 0,Y 100.494,Z 698.26,A -85,B 0,C 180,E1 -27762.752,E2 -27762.752} C_VEL
LIN {X 0,Y 96.148,Z 709.487,A -85,B 0,C 180,E1 -27766.021,E2 -27766.021} C_VEL
LIN {X 0,Y 91.654,Z 719.689,A -85,B 0,C 180,E1 -27770.07,E2 -27770.07} C_VEL
LIN {X 0,Y 86.876,Z 729.632,A -85,B 0,C 180,E1 -27775.51,E2 -27775.51} C_VEL
LIN {X 0,Y 82.724,Z 738.42,A -85,B 0,C 180,E1 -27782.144,E2 -27782.144} C_VEL
LIN {X 0,Y 79.701,Z 745.385,A -85,B 0,C 180,E1 -27789.347,E2 -27789.347} C_VEL
LIN {X 0,Y 77.9,Z 750.92,A -85,B 0,C 180,E1 -27796.965,E2 -27796.965} C_VEL
LIN {X 0,Y 77.486,Z 755.861,A -85,B 0,C 180,E1 -27806.155,E2 -27806.155} C_VEL
LIN {X 0,Y 77.611,Z 757.439,A -85,B 0,C 180,E1 -27810,E2 -27810} C_VEL
LIN {X 0,Y 77.294,Z 759.09,A -85,B 0,C 180,E1 -27815.217,E2 -27815.217} C_VEL
LIN {X 0,Y 78.113,Z 761.113,A -85,B 0,C 180,E1 -27825.659,E2 -27825.659} C_VEL
LIN {X 0,Y 81.357,Z 761.671,A -85,B 0,C 180,E1 -27835.589,E2 -27835.589} C_VEL
LIN {X 0,Y 87.067,Z 760.812,A -85,B 0,C 180,E1 -27844.404,E2 -27844.404} C_VEL
LIN {X 0,Y 94.671,Z 758.448,A -85,B 0,C 180,E1 -27851.921,E2 -27851.921} C_VEL
LIN {X 0,Y 103.672,Z 754.602,A -85,B 0,C 180,E1 -27858.218,E2 -27858.218} C_VEL
LIN {X 0,Y 111.268,Z 750.607,A -85,B 0,C 180,E1 -27862.14,E2 -27862.14} C_VEL
LIN {X 0,Y 119.384,Z 745.577,A -85,B 0,C 180,E1 -27865.501,E2 -27865.501} C_VEL
LIN {X 0,Y 129.38,Z 738.199,A -85,B 0,C 180,E1 -27868.818,E2 -27868.818} C_VEL
LIN {X 0,Y 138.307,Z 730.343,A -85,B 0,C 180,E1 -27871.226,E2 -27871.226} C_VEL
LIN {X 0,Y 147.53,Z 720.702,A -85,B 0,C 180,E1 -27873.276,E2 -27873.276} C_VEL
LIN {X 0,Y 155.405,Z 710.79,A -85,B 0,C 180,E1 -27874.75,E2 -27874.75} C_VEL
LIN {X 0,Y 162.619,Z 699.751,A -85,B 0,C 180,E1 -27875.916,E2 -27875.916} C_VEL
LIN {X 0,Y 168.342,Z 689.062,A -85,B 0,C 180,E1 -27876.699,E2 -27876.699} C_VEL
LIN {X 0,Y 173.274,Z 677.535,A -85,B 0,C 180,E1 -27877.328,E2 -27877.328} C_VEL
LIN {X 0,Y 177.382,Z 664.652,A -85,B 0,C 180,E1 -27877.925,E2 -27877.925} C_VEL
LIN {X 0,Y 177.469,Z 663.179,A -85,B 0,C 180,E1 -27879.375,E2 -27879.375} C_VEL
LIN {X 0,Y 177.503,Z 662.117,A -85,B 0,C 180,E1 -27881.847,E2 -27881.847} C_VEL
LIN {X 0,Y 177.791,Z 662.438,A -85,B 0,C 180,E1 -27884.98,E2 -27884.98} C_VEL
LIN {X 0,Y 175.856,Z 669.2,A -85,B 0,C 180,E1 -27885.324,E2 -27885.324} C_VEL
LIN {X 0,Y 173.963,Z 674.788,A -85,B 0,C 180,E1 -27885.451,E2 -27885.451} C_VEL
LIN {X 0,Y 170.083,Z 683.866,A -85,B 0,C 180,E1 -27885.144,E2 -27885.144} C_VEL
LIN {X 0,Y 165.528,Z 692.6,A -85,B 0,C 180,E1 -27884.891,E2 -27884.891} C_VEL
LIN {X 0,Y 162.569,Z 697.642,A -85,B 0,C 180,E1 -27885.129,E2 -27885.129} C_VEL
LIN {X 0,Y 155.14,Z 708.631,A -85,B 0,C 180,E1 -27886.462,E2 -27886.462} C_VEL
LIN {X 0,Y 147.27,Z 718.114,A -85,B 0,C 180,E1 -27888.028,E2 -27888.028} C_VEL
LIN {X 0,Y 139.231,Z 726.23,A -85,B 0,C 180,E1 -27889.829,E2 -27889.829} C_VEL
LIN {X 0,Y 129.397,Z 734.458,A -85,B 0,C 180,E1 -27892.393,E2 -27892.393} C_VEL
LIN {X 0,Y 119.857,Z 741.001,A -85,B 0,C 180,E1 -27895.414,E2 -27895.414} C_VEL
LIN {X 0,Y 110.075,Z 746.373,A -85,B 0,C 180,E1 -27899.18,E2 -27899.18} C_VEL
LIN {X 0,Y 100.29,Z 750.601,A -85,B 0,C 180,E1 -27904.016,E2 -27904.016} C_VEL
LIN {X 0,Y 92.51,Z 753.076,A -85,B 0,C 180,E1 -27909.036,E2 -27909.036} C_VEL
LIN {X 0,Y 86.395,Z 754.386,A -85,B 0,C 180,E1 -27914.123,E2 -27914.123} C_VEL
LIN {X 0,Y 80.641,Z 754.966,A -85,B 0,C 180,E1 -27920.399,E2 -27920.399} C_VEL
LIN {X 0,Y 75.917,Z 754.674,A -85,B 0,C 180,E1 -27927.57,E2 -27927.57} C_VEL
LIN {X 0,Y 71.556,Z 752.877,A -85,B 0,C 180,E1 -27938.213,E2 -27938.213} C_VEL
LIN {X 0,Y 69.706,Z 749.749,A -85,B 0,C 180,E1 -27949.055,E2 -27949.055} C_VEL
LIN {X 0,Y 70.116,Z 745.096,A -85,B 0,C 180,E1 -27959.923,E2 -27959.923} C_VEL
LIN {X 0,Y 71.884,Z 740.069,A -85,B 0,C 180,E1 -27968.494,E2 -27968.494} C_VEL
LIN {X 0,Y 74.743,Z 733.875,A -85,B 0,C 180,E1 -27976.405,E2 -27976.405} C_VEL
LIN {X 0,Y 78.699,Z 726.112,A -85,B 0,C 180,E1 -27983.783,E2 -27983.783} C_VEL
LIN {X 0,Y 83.282,Z 717.122,A -85,B 0,C 180,E1 -27990,E2 -27990} C_VEL
LIN {X 0,Y 88.219,Z 706.911,A -85,B 0,C 180,E1 -27995.142,E2 -27995.142} C_VEL
LIN {X 0,Y 92.799,Z 696.344,A -85,B 0,C 180,E1 -27999.045,E2 -27999.045} C_VEL
LIN {X 0,Y 96.907,Z 685.29,A -85,B 0,C 180,E1 -28002.034,E2 -28002.034} C_VEL
LIN {X 0,Y 100.884,Z 672.016,A -85,B 0,C 180,E1 -28004.634,E2 -28004.634} C_VEL
LIN {X 0,Y 103.755,Z 659.036,A -85,B 0,C 180,E1 -28006.384,E2 -28006.384} C_VEL
LIN {X 0,Y 105.843,Z 644.884,A -85,B 0,C 180,E1 -28007.577,E2 -28007.577} C_VEL
LIN {X 0,Y 108.686,Z 617.679,A -85,B 0,C 180,E1 -28009.105,E2 -28009.105} C_VEL
LIN {X 0,Y 107.169,Z 613.938,A -85,B 0,C 180,E1 -28010.306,E2 -28010.306} C_VEL
LIN {X 0,Y 101.775,Z 602.16,A -85,B 0,C 180,E1 -28014.927,E2 -28014.927} C_VEL
LIN {X 0,Y 96.439,Z 592.675,A -85,B 0,C 180,E1 -28020.054,E2 -28020.054} C_VEL
LIN {X 0,Y 91.995,Z 585.632,A -85,B 0,C 180,E1 -28025.206,E2 -28025.206} C_VEL
LIN {X 0,Y 89.088,Z 581.453,A -85,B 0,C 180,E1 -28029.131,E2 -28029.131} C_VEL
LIN {X 0,Y 86.655,Z 577.832,A -85,B 0,C 180,E1 -28033.123,E2 -28033.123} C_VEL
LIN {X 0,Y 86.122,Z 577.096,A -85,B 0,C 180,E1 -28034.094,E2 -28034.094} C_VEL
LIN {X 0,Y 83.783,Z 574.545,A -85,B 0,C 180,E1 -28038.672,E2 -28038.672} C_VEL
LIN {X 0,Y 82.848,Z 572.361,A -85,B 0,C 180,E1 -28041.275,E2 -28041.275} C_VEL
LIN {X 0,Y 79.318,Z 569.2,A -85,B 0,C 180,E1 -28056.504,E2 -28056.504} C_VEL
LIN {X 0,Y 79.55,Z 568.911,A -85,B 0,C 180,E1 -28066.358,E2 -28066.358} C_VEL
LIN {X 0,Y 83.273,Z 572.027,A -85,B 0,C 180,E1 -28080.512,E2 -28080.512} C_VEL
LIN {X 0,Y 84.895,Z 575.326,A -85,B 0,C 180,E1 -28084.506,E2 -28084.506} C_VEL
LIN {X 0,Y 86.79,Z 577.42,A -85,B 0,C 180,E1 -28088.003,E2 -28088.003} C_VEL
LIN {X 0,Y 89.076,Z 581.096,A -85,B 0,C 180,E1 -28091.775,E2 -28091.775} C_VEL
LIN {X 0,Y 92.629,Z 586.604,A -85,B 0,C 180,E1 -28096.603,E2 -28096.603} C_VEL
LIN {X 0,Y 96.416,Z 592.884,A -85,B 0,C 180,E1 -28100.96,E2 -28100.96} C_VEL
LIN {X 0,Y 100.002,Z 599.586,A -85,B 0,C 180,E1 -28104.544,E2 -28104.544} C_VEL
LIN {X 0,Y 103.723,Z 610.241,A -85,B 0,C 180,E1 -28108.316,E2 -28108.316} C_VEL
LIN {X 0,Y 107.561,Z 623.329,A -85,B 0,C 180,E1 -28111.929,E2 -28111.929} C_VEL
LIN {X 0,Y 107.839,Z 626.267,A -85,B 0,C 180,E1 -28112.388,E2 -28112.388} C_VEL
LIN {X 0,Y 107.763,Z 631.483,A -85,B 0,C 180,E1 -28112.911,E2 -28112.911} C_VEL
LIN {X 0,Y 104.592,Z 660.478,A -85,B 0,C 180,E1 -28114.657,E2 -28114.657} C_VEL
LIN {X 0,Y 102.257,Z 673.099,A -85,B 0,C 180,E1 -28115.934,E2 -28115.934} C_VEL
LIN {X 0,Y 98.871,Z 685.591,A -85,B 0,C 180,E1 -28117.742,E2 -28117.742} C_VEL
LIN {X 0,Y 94.631,Z 698.024,A -85,B 0,C 180,E1 -28120.428,E2 -28120.428} C_VEL
LIN {X 0,Y 90.062,Z 709.195,A -85,B 0,C 180,E1 -28123.796,E2 -28123.796} C_VEL
LIN {X 0,Y 85.381,Z 719.215,A -85,B 0,C 180,E1 -28127.947,E2 -28127.947} C_VEL
LIN {X 0,Y 80.258,Z 729.264,A -85,B 0,C 180,E1 -28133.767,E2 -28133.767} C_VEL
LIN {X 0,Y 75.852,Z 738.043,A -85,B 0,C 180,E1 -28140.895,E2 -28140.895} C_VEL
LIN {X 0,Y 72.631,Z 744.993,A -85,B 0,C 180,E1 -28148.725,E2 -28148.725} C_VEL
LIN {X 0,Y 70.637,Z 751.33,A -85,B 0,C 180,E1 -28158.522,E2 -28158.522} C_VEL
LIN {X 0,Y 70.432,Z 755.057,A -85,B 0,C 180,E1 -28166.275,E2 -28166.275} C_VEL
LIN {X 0,Y 70.542,Z 756.509,A -85,B 0,C 180,E1 -28170,E2 -28170} C_VEL
LIN {X 0,Y 70.242,Z 758.244,A -85,B 0,C 180,E1 -28175.742,E2 -28175.742} C_VEL
LIN {X 0,Y 71.283,Z 760.488,A -85,B 0,C 180,E1 -28187.204,E2 -28187.204} C_VEL
LIN {X 0,Y 74.992,Z 761.214,A -85,B 0,C 180,E1 -28197.942,E2 -28197.942} C_VEL
LIN {X 0,Y 81.289,Z 760.541,A -85,B 0,C 180,E1 -28207.242,E2 -28207.242} C_VEL
LIN {X 0,Y 89.502,Z 758.436,A -85,B 0,C 180,E1 -28214.967,E2 -28214.967} C_VEL
LIN {X 0,Y 99.085,Z 754.791,A -85,B 0,C 180,E1 -28221.279,E2 -28221.279} C_VEL
LIN {X 0,Y 107.065,Z 750.997,A -85,B 0,C 180,E1 -28225.136,E2 -28225.136} C_VEL
LIN {X 0,Y 115.539,Z 746.199,A -85,B 0,C 180,E1 -28228.383,E2 -28228.383} C_VEL
LIN {X 0,Y 125.888,Z 739.167,A -85,B 0,C 180,E1 -28231.554,E2 -28231.554} C_VEL
LIN {X 0,Y 135.079,Z 731.668,A -85,B 0,C 180,E1 -28233.828,E2 -28233.828} C_VEL
LIN {X 0,Y 142.935,Z 724.097,A -85,B 0,C 180,E1 -28235.451,E2 -28235.451} C_VEL
LIN {X 0,Y 151.768,Z 713.985,A -85,B 0,C 180,E1 -28236.976,E2 -28236.976} C_VEL
LIN {X 0,Y 159.916,Z 702.654,A -85,B 0,C 180,E1 -28238.183,E2 -28238.183} C_VEL
LIN {X 0,Y 166.329,Z 691.691,A -85,B 0,C 180,E1 -28238.979,E2 -28238.979} C_VEL
LIN {X 0,Y 171.96,Z 679.436,A -85,B 0,C 180,E1 -28239.607,E2 -28239.607} C_VEL
LIN {X 0,Y 175.197,Z 670.589,A -85,B 0,C 180,E1 -28239.961,E2 -28239.961} C_VEL
LIN {X 0,Y 175.484,Z 669.329,A -85,B 0,C 180,E1 -28240.826,E2 -28240.826} C_VEL
LIN {X 0,Y 175.59,Z 668.944,A -85,B 0,C 180,E1 -28242.925,E2 -28242.925} C_VEL
LIN {X 0,Y 170.858,Z 681.618,A -85,B 0,C 180,E1 -28243.732,E2 -28243.732} C_VEL
LIN {X 0,Y 164.955,Z 693.545,A -85,B 0,C 180,E1 -28244.712,E2 -28244.712} C_VEL
LIN {X 0,Y 162.569,Z 697.642,A -85,B 0,C 180,E1 -28245.129,E2 -28245.129} C_VEL
LIN {X 0,Y 159.389,Z 702.6,A -85,B 0,C 180,E1 -28245.414,E2 -28245.414} C_VEL
LIN {X 0,Y 153.493,Z 710.547,A -85,B 0,C 180,E1 -28245.367,E2 -28245.367} C_VEL
LIN {X 0,Y 147.053,Z 718.008,A -85,B 0,C 180,E1 -28245.412,E2 -28245.412} C_VEL
LIN {X 0,Y 143.03,Z 722.115,A -85,B 0,C 180,E1 -28245.885,E2 -28245.885} C_VEL
LIN {X 0,Y 133.618,Z 730.542,A -85,B 0,C 180,E1 -28247.853,E2 -28247.853} C_VEL
LIN {X 0,Y 124.108,Z 737.578,A -85,B 0,C 180,E1 -28250.217,E2 -28250.217} C_VEL
LIN {X 0,Y 113.163,Z 744.164,A -85,B 0,C 180,E1 -28253.545,E2 -28253.545} C_VEL
LIN {X 0,Y 101.973,Z 749.33,A -85,B 0,C 180,E1 -28257.878,E2 -28257.878} C_VEL
LIN {X 0,Y 91.513,Z 752.875,A -85,B 0,C 180,E1 -28263.298,E2 -28263.298} C_VEL
LIN {X 0,Y 82.329,Z 754.827,A -85,B 0,C 180,E1 -28269.828,E2 -28269.828} C_VEL
LIN {X 0,Y 74.046,Z 755.426,A -85,B 0,C 180,E1 -28278.356,E2 -28278.356} C_VEL
LIN {X 0,Y 69.694,Z 754.989,A -85,B 0,C 180,E1 -28284.831,E2 -28284.831} C_VEL
LIN {X 0,Y 66.299,Z 753.956,A -85,B 0,C 180,E1 -28292.003,E2 -28292.003} C_VEL
LIN {X 0,Y 63.541,Z 751.78,A -85,B 0,C 180,E1 -28301.573,E2 -28301.573} C_VEL
LIN {X 0,Y 62.504,Z 748.504,A -85,B 0,C 180,E1 -28311.909,E2 -28311.909} C_VEL
LIN {X 0,Y 63.554,Z 743.279,A -85,B 0,C 180,E1 -28323.748,E2 -28323.748} C_VEL
LIN {X 0,Y 66.06,Z 737.516,A -85,B 0,C 180,E1 -28333.224,E2 -28333.224} C_VEL
LIN {X 0,Y 70.133,Z 729.731,A -85,B 0,C 180,E1 -28342.519,E2 -28342.519} C_VEL
LIN {X 0,Y 75.045,Z 720.788,A -85,B 0,C 180,E1 -28350,E2 -28350} C_VEL
LIN {X 0,Y 80.088,Z 711.337,A -85,B 0,C 180,E1 -28355.665,E2 -28355.665} C_VEL
LIN {X 0,Y 85.303,Z 700.51,A -85,B 0,C 180,E1 -28360.31,E2 -28360.31} C_VEL
LIN {X 0,Y 90.366,Z 688.176,A -85,B 0,C 180,E1 -28364.066,E2 -28364.066} C_VEL
LIN {X 0,Y 94.509,Z 675.72,A -85,B 0,C 180,E1 -28366.747,E2 -28366.747} C_VEL
LIN {X 0,Y 97.957,Z 662.008,A -85,B 0,C 180,E1 -28368.779,E2 -28368.779} C_VEL
LIN {X 0,Y 100.185,Z 648.902,A -85,B 0,C 180,E1 -28370.048,E2 -28370.048} C_VEL
LIN {X 0,Y 103.399,Z 619.469,A -85,B 0,C 180,E1 -28371.779,E2 -28371.779} C_VEL
LIN {X 0,Y 97.785,Z 606.795,A -85,B 0,C 180,E1 -28377.009,E2 -28377.009} C_VEL
LIN {X 0,Y 92.794,Z 597.513,A -85,B 0,C 180,E1 -28382.44,E2 -28382.44} C_VEL
LIN {X 0,Y 89.092,Z 591.374,A -85,B 0,C 180,E1 -28387.19,E2 -28387.19} C_VEL
LIN {X 0,Y 86.701,Z 587.631,A -85,B 0,C 180,E1 -28390.828,E2 -28390.828} C_VEL
LIN {X 0,Y 84.055,Z 583.584,A -85,B 0,C 180,E1 -28395.691,E2 -28395.691} C_VEL
LIN {X 0,Y 81.773,Z 580.643,A -85,B 0,C 180,E1 -28400.801,E2 -28400.801} C_VEL
LIN {X 0,Y 81.182,Z 579.164,A -85,B 0,C 180,E1 -28402.703,E2 -28402.703} C_VEL
LIN {X 0,Y 78.219,Z 576.111,A -85,B 0,C 180,E1 -28417.554,E2 -28417.554} C_VEL
LIN {X 0,Y 78.385,Z 575.866,A -85,B 0,C 180,E1 -28425.27,E2 -28425.27} C_VEL
LIN {X 0,Y 81.557,Z 578.818,A -85,B 0,C 180,E1 -28439.077,E2 -28439.077} C_VEL
LIN {X 0,Y 83.36,Z 582.233,A -85,B 0,C 180,E1 -28443.737,E2 -28443.737} C_VEL
LIN {X 0,Y 84.713,Z 583.98,A -85,B 0,C 180,E1 -28446.477,E2 -28446.477} C_VEL
LIN {X 0,Y 87.68,Z 588.957,A -85,B 0,C 180,E1 -28451.69,E2 -28451.69} C_VEL
LIN {X 0,Y 90.231,Z 593.169,A -85,B 0,C 180,E1 -28455.315,E2 -28455.315} C_VEL
LIN {X 0,Y 94.172,Z 600.26,A -85,B 0,C 180,E1 -28460.225,E2 -28460.225} C_VEL
LIN {X 0,Y 96.307,Z 604.73,A -85,B 0,C 180,E1 -28462.598,E2 -28462.598} C_VEL
LIN {X 0,Y 99.51,Z 614.588,A -85,B 0,C 180,E1 -28466.196,E2 -28466.196} C_VEL
LIN {X 0,Y 102.667,Z 626.292,A -85,B 0,C 180,E1 -28469.616,E2 -28469.616} C_VEL
LIN {X 0,Y 102.643,Z 631.568,A -85,B 0,C 180,E1 -28470.228,E2 -28470.228} C_VEL
LIN {X 0,Y 99.4,Z 660.029,A -85,B 0,C 180,E1 -28471.958,E2 -28471.958} C_VEL
LIN {X 0,Y 96.904,Z 672.825,A -85,B 0,C 180,E1 -28473.25,E2 -28473.25} C_VEL
LIN {X 0,Y 93.376,Z 685.281,A -85,B 0,C 180,E1 -28475.066,E2 -28475.066} C_VEL
LIN {X 0,Y 88.947,Z 697.702,A -85,B 0,C 180,E1 -28477.803,E2 -28477.803} C_VEL
LIN {X 0,Y 84.119,Z 708.847,A -85,B 0,C 180,E1 -28481.243,E2 -28481.243} C_VEL
LIN {X 0,Y 79.176,Z 718.834,A -85,B 0,C 180,E1 -28485.547,E2 -28485.547} C_VEL
LIN {X 0,Y 73.735,Z 728.898,A -85,B 0,C 180,E1 -28491.718,E2 -28491.718} C_VEL
LIN {X 0,Y 69.002,Z 737.66,A -85,B 0,C 180,E1 -28499.386,E2 -28499.386} C_VEL
LIN {X 0,Y 65.594,Z 744.606,A -85,B 0,C 180,E1 -28507.976,E2 -28507.976} C_VEL
LIN {X 0,Y 63.677,Z 750.115,A -85,B 0,C 180,E1 -28517.248,E2 -28517.248} C_VEL
LIN {X 0,Y 63.374,Z 754.263,A -85,B 0,C 180,E1 -28526.494,E2 -28526.494} C_VEL
LIN {X 0,Y 63.492,Z 755.561,A -85,B 0,C 180,E1 -28530,E2 -28530} C_VEL
LIN {X 0,Y 63.22,Z 757.369,A -85,B 0,C 180,E1 -28536.382,E2 -28536.382} C_VEL
LIN {X 0,Y 64.526,Z 759.789,A -85,B 0,C 180,E1 -28549.071,E2 -28549.071} C_VEL
LIN {X 0,Y 68.782,Z 760.754,A -85,B 0,C 180,E1 -28560.722,E2 -28560.722} C_VEL
LIN {X 0,Y 75.744,Z 760.263,A -85,B 0,C 180,E1 -28570.503,E2 -28570.503} C_VEL
LIN {X 0,Y 84.61,Z 758.367,A -85,B 0,C 180,E1 -28578.379,E2 -28578.379} C_VEL
LIN {X 0,Y 89.546,Z 756.879,A -85,B 0,C 180,E1 -28581.705,E2 -28581.705} C_VEL
LIN {X 0,Y 100.332,Z 752.694,A -85,B 0,C 180,E1 -28587.198,E2 -28587.198} C_VEL
LIN {X 0,Y 108.981,Z 748.481,A -85,B 0,C 180,E1 -28590.525,E2 -28590.525} C_VEL
LIN {X 0,Y 119.609,Z 742.18,A -85,B 0,C 180,E1 -28593.643,E2 -28593.643} C_VEL
LIN {X 0,Y 128.959,Z 735.45,A -85,B 0,C 180,E1 -28595.897,E2 -28595.897} C_VEL
LIN {X 0,Y 138.562,Z 727.268,A -85,B 0,C 180,E1 -28597.765,E2 -28597.765} C_VEL
LIN {X 0,Y 146.711,Z 718.974,A -85,B 0,C 180,E1 -28599.083,E2 -28599.083} C_VEL
LIN {X 0,Y 154.97,Z 708.881,A -85,B 0,C 180,E1 -28600.221,E2 -28600.221} C_VEL
LIN {X 0,Y 162.497,Z 697.672,A -85,B 0,C 180,E1 -28601.098,E2 -28601.098} C_VEL
LIN {X 0,Y 166.108,Z 691.34,A -85,B 0,C 180,E1 -28601.445,E2 -28601.445} C_VEL
LIN {X 0,Y 166.892,Z 689.74,A -85,B 0,C 180,E1 -28601.898,E2 -28601.898} C_VEL
LIN {X 0,Y 160.944,Z 699.991,A -85,B 0,C 180,E1 -28602.784,E2 -28602.784} C_VEL
LIN {X 0,Y 153.236,Z 710.729,A -85,B 0,C 180,E1 -28604.026,E2 -28604.026} C_VEL
LIN {X 0,Y 145.21,Z 719.88,A -85,B 0,C 180,E1 -28605.455,E2 -28605.455} C_VEL
LIN {X 0,Y 143.03,Z 722.115,A -85,B 0,C 180,E1 -28605.885,E2 -28605.885} C_VEL
LIN {X 0,Y 138.787,Z 726.109,A -85,B 0,C 180,E1 -28606.42,E2 -28606.42} C_VEL
LIN {X 0,Y 127.949,Z 734.737,A -85,B 0,C 180,E1 -28606.822,E2 -28606.822} C_VEL
LIN {X 0,Y 121.494,Z 739.048,A -85,B 0,C 180,E1 -28607.385,E2 -28607.385} C_VEL
LIN {X 0,Y 118.35,Z 740.921,A -85,B 0,C 180,E1 -28608.015,E2 -28608.015} C_VEL
LIN {X 0,Y 106.609,Z 746.992,A -85,B 0,C 180,E1 -28611.424,E2 -28611.424} C_VEL
LIN {X 0,Y 95.178,Z 751.43,A -85,B 0,C 180,E1 -28615.763,E2 -28615.763} C_VEL
LIN {X 0,Y 84.358,Z 754.341,A -85,B 0,C 180,E1 -28621.378,E2 -28621.378} C_VEL
LIN {X 0,Y 77.723,Z 755.409,A -85,B 0,C 180,E1 -28625.935,E2 -28625.935} C_VEL
LIN {X 0,Y 71.669,Z 755.873,A -85,B 0,C 180,E1 -28631.307,E2 -28631.307} C_VEL
LIN {X 0,Y 65.433,Z 755.609,A -85,B 0,C 180,E1 -28638.794,E2 -28638.794} C_VEL
LIN {X 0,Y 60.494,Z 754.43,A -85,B 0,C 180,E1 -28647.687,E2 -28647.687} C_VEL
LIN {X 0,Y 57.063,Z 752.291,A -85,B 0,C 180,E1 -28658.006,E2 -28658.006} C_VEL
LIN {X 0,Y 55.426,Z 748.699,A -85,B 0,C 180,E1 -28670.655,E2 -28670.655} C_VEL
LIN {X 0,Y 56.032,Z 744.61,A -85,B 0,C 180,E1 -28681.395,E2 -28681.395} C_VEL
LIN {X 0,Y 58.705,Z 738.394,A -85,B 0,C 180,E1 -28693.271,E2 -28693.271} C_VEL
LIN {X 0,Y 62.897,Z 730.754,A -85,B 0,C 180,E1 -28703.585,E2 -28703.585} C_VEL
LIN {X 0,Y 67.768,Z 722.537,A -85,B 0,C 180,E1 -28711.333,E2 -28711.333} C_VEL
LIN {X 0,Y 73.206,Z 713.077,A -85,B 0,C 180,E1 -28717.585,E2 -28717.585} C_VEL
LIN {X 0,Y 78.878,Z 702.113,A -85,B 0,C 180,E1 -28722.718,E2 -28722.718} C_VEL
LIN {X 0,Y 83.951,Z 690.757,A -85,B 0,C 180,E1 -28726.411,E2 -28726.411} C_VEL
LIN {X 0,Y 88.224,Z 679.181,A -85,B 0,C 180,E1 -28729.118,E2 -28729.118} C_VEL
LIN {X 0,Y 92.019,Z 666.116,A -85,B 0,C 180,E1 -28731.252,E2 -28731.252} C_VEL
LIN {X 0,Y 94.785,Z 652.031,A -85,B 0,C 180,E1 -28732.784,E2 -28732.784} C_VEL
LIN {X 0,Y 98.339,Z 621.972,A -85,B 0,C 180,E1 -28734.609,E2 -28734.609} C_VEL
LIN {X 0,Y 94.107,Z 611.815,A -85,B 0,C 180,E1 -28739.073,E2 -28739.073} C_VEL
LIN {X 0,Y 89.65,Z 603.002,A -85,B 0,C 180,E1 -28744.491,E2 -28744.491} C_VEL
LIN {X 0,Y 86.501,Z 597.381,A -85,B 0,C 180,E1 -28749.004,E2 -28749.004} C_VEL
LIN {X 0,Y 84.226,Z 593.566,A -85,B 0,C 180,E1 -28752.92,E2 -28752.92} C_VEL
LIN {X 0,Y 81.988,Z 589.963,A -85,B 0,C 180,E1 -28757.471,E2 -28757.471} C_VEL
LIN {X 0,Y 79.832,Z 586.621,A -85,B 0,C 180,E1 -28763.209,E2 -28763.209} C_VEL
LIN {X 0,Y 79.502,Z 585.856,A -85,B 0,C 180,E1 -28764.426,E2 -28764.426} C_VEL
LIN {X 0,Y 77.182,Z 583.196,A -85,B 0,C 180,E1 -28777.235,E2 -28777.235} C_VEL
LIN {X 0,Y 77.37,Z 582.97,A -85,B 0,C 180,E1 -28785.695,E2 -28785.695} C_VEL
LIN {X 0,Y 79.965,Z 585.703,A -85,B 0,C 180,E1 -28797.799,E2 -28797.799} C_VEL
LIN {X 0,Y 81.805,Z 589.113,A -85,B 0,C 180,E1 -28802.908,E2 -28802.908} C_VEL
LIN {X 0,Y 82.782,Z 590.639,A -85,B 0,C 180,E1 -28805.049,E2 -28805.049} C_VEL
LIN {X 0,Y 85.251,Z 595.058,A -85,B 0,C 180,E1 -28809.895,E2 -28809.895} C_VEL
LIN {X 0,Y 88.657,Z 601.146,A -85,B 0,C 180,E1 -28815.134,E2 -28815.134} C_VEL
LIN {X 0,Y 92.229,Z 608.476,A -85,B 0,C 180,E1 -28819.844,E2 -28819.844} C_VEL
LIN {X 0,Y 95.23,Z 618.434,A -85,B 0,C 180,E1 -28823.741,E2 -28823.741} C_VEL
LIN {X 0,Y 97.867,Z 628.75,A -85,B 0,C 180,E1 -28826.958,E2 -28826.958} C_VEL
LIN {X 0,Y 97.386,Z 634.934,A -85,B 0,C 180,E1 -28827.451,E2 -28827.451} C_VEL
LIN {X 0,Y 94.396,Z 659.837,A -85,B 0,C 180,E1 -28828.984,E2 -28828.984} C_VEL
LIN {X 0,Y 91.71,Z 672.865,A -85,B 0,C 180,E1 -28830.296,E2 -28830.296} C_VEL
LIN {X 0,Y 88.112,Z 684.97,A -85,B 0,C 180,E1 -28832.064,E2 -28832.064} C_VEL
LIN {X 0,Y 83.461,Z 697.345,A -85,B 0,C 180,E1 -28834.815,E2 -28834.815} C_VEL
LIN {X 0,Y 78.385,Z 708.468,A -85,B 0,C 180,E1 -28838.328,E2 -28838.328} C_VEL
LIN {X 0,Y 73.085,Z 718.52,A -85,B 0,C 180,E1 -28842.822,E2 -28842.822} C_VEL
LIN {X 0,Y 67.319,Z 728.461,A -85,B 0,C 180,E1 -28849.272,E2 -28849.272} C_VEL
LIN {X 0,Y 62.24,Z 737.211,A -85,B 0,C 180,E1 -28857.565,E2 -28857.565} C_VEL
LIN {X 0,Y 58.568,Z 744.143,A -85,B 0,C 180,E1 -28867.047,E2 -28867.047} C_VEL
LIN {X 0,Y 56.449,Z 750.46,A -85,B 0,C 180,E1 -28879.237,E2 -28879.237} C_VEL
LIN {X 0,Y 56.431,Z 754.52,A -85,B 0,C 180,E1 -28890,E2 -28890} C_VEL
LIN {X 0,Y 56.199,Z 756.477,A -85,B 0,C 180,E1 -28897.184,E2 -28897.184} C_VEL
LIN {X 0,Y 57.863,Z 759.073,A -85,B 0,C 180,E1 -28911.369,E2 -28911.369} C_VEL
LIN {X 0,Y 62.77,Z 760.218,A -85,B 0,C 180,E1 -28924.042,E2 -28924.042} C_VEL
LIN {X 0,Y 70.485,Z 759.982,A -85,B 0,C 180,E1 -28934.262,E2 -28934.262} C_VEL
LIN {X 0,Y 80.049,Z 758.28,A -85,B 0,C 180,E1 -28942.199,E2 -28942.199} C_VEL
LIN {X 0,Y 90.882,Z 755.155,A -85,B 0,C 180,E1 -28948.279,E2 -28948.279} C_VEL
LIN {X 0,Y 99.655,Z 751.767,A -85,B 0,C 180,E1 -28951.827,E2 -28951.827} C_VEL
LIN {X 0,Y 108.807,Z 747.412,A -85,B 0,C 180,E1 -28954.724,E2 -28954.724} C_VEL
LIN {X 0,Y 119.835,Z 741.022,A -85,B 0,C 180,E1 -28957.469,E2 -28957.469} C_VEL
LIN {X 0,Y 129.515,Z 734.182,A -85,B 0,C 180,E1 -28959.396,E2 -28959.396} C_VEL
LIN {X 0,Y 139.375,Z 725.758,A -85,B 0,C 180,E1 -28960.987,E2 -28960.987} C_VEL
LIN {X 0,Y 147.696,Z 717.247,A -85,B 0,C 180,E1 -28962.112,E2 -28962.112} C_VEL
LIN {X 0,Y 139.236,Z 725.628,A -85,B 0,C 180,E1 -28963.538,E2 -28963.538} C_VEL
LIN {X 0,Y 130.887,Z 732.543,A -85,B 0,C 180,E1 -28965.125,E2 -28965.125} C_VEL
LIN {X 0,Y 120.6,Z 739.588,A -85,B 0,C 180,E1 -28967.446,E2 -28967.446} C_VEL
LIN {X 0,Y 118.35,Z 740.921,A -85,B 0,C 180,E1 -28968.015,E2 -28968.015} C_VEL
LIN {X 0,Y 113.448,Z 743.654,A -85,B 0,C 180,E1 -28968.962,E2 -28968.962} C_VEL
LIN {X 0,Y 104.596,Z 747.8,A -85,B 0,C 180,E1 -28969.865,E2 -28969.865} C_VEL
LIN {X 0,Y 95.546,Z 751.205,A -85,B 0,C 180,E1 -28971.033,E2 -28971.033} C_VEL
LIN {X 0,Y 90.413,Z 752.704,A -85,B 0,C 180,E1 -28972.539,E2 -28972.539} C_VEL
LIN {X 0,Y 84.422,Z 754.242,A -85,B 0,C 180,E1 -28975.222,E2 -28975.222} C_VEL
LIN {X 0,Y 75.841,Z 755.728,A -85,B 0,C 180,E1 -28979.997,E2 -28979.997} C_VEL
LIN {X 0,Y 67.972,Z 756.331,A -85,B 0,C 180,E1 -28985.932,E2 -28985.932} C_VEL
LIN {X 0,Y 60.921,Z 756.07,A -85,B 0,C 180,E1 -28993.336,E2 -28993.336} C_VEL
LIN {X 0,Y 54.116,Z 754.54,A -85,B 0,C 180,E1 -29004.625,E2 -29004.625} C_VEL
LIN {X 0,Y 49.606,Z 751.571,A -85,B 0,C 180,E1 -29018.813,E2 -29018.813} C_VEL
LIN {X 0,Y 48.348,Z 747.161,A -85,B 0,C 180,E1 -29034.448,E2 -29034.448} C_VEL
LIN {X 0,Y 49.759,Z 742.293,A -85,B 0,C 180,E1 -29047.108,E2 -29047.108} C_VEL
LIN {X 0,Y 52.975,Z 736.246,A -85,B 0,C 180,E1 -29058.522,E2 -29058.522} C_VEL
LIN {X 0,Y 57.42,Z 729.049,A -85,B 0,C 180,E1 -29068.15,E2 -29068.15} C_VEL
LIN {X 0,Y 63.146,Z 720.068,A -85,B 0,C 180,E1 -29076.39,E2 -29076.39} C_VEL
LIN {X 0,Y 68.985,Z 710.339,A -85,B 0,C 180,E1 -29082.438,E2 -29082.438} C_VEL
LIN {X 0,Y 74.749,Z 699.497,A -85,B 0,C 180,E1 -29087.086,E2 -29087.086} C_VEL
LIN {X 0,Y 80.002,Z 687.888,A -85,B 0,C 180,E1 -29090.572,E2 -29090.572} C_VEL
LIN {X 0,Y 84.425,Z 675.602,A -85,B 0,C 180,E1 -29093.151,E2 -29093.151} C_VEL
LIN {X 0,Y 88.11,Z 662.152,A -85,B 0,C 180,E1 -29095.083,E2 -29095.083} C_VEL
LIN {X 0,Y 90.471,Z 649.454,A -85,B 0,C 180,E1 -29096.251,E2 -29096.251} C_VEL
LIN {X 0,Y 93.463,Z 624.346,A -85,B 0,C 180,E1 -29097.728,E2 -29097.728} C_VEL
LIN {X 0,Y 90.261,Z 616.13,A -85,B 0,C 180,E1 -29101.691,E2 -29101.691} C_VEL
LIN {X 0,Y 86.357,Z 607.981,A -85,B 0,C 180,E1 -29107.041,E2 -29107.041} C_VEL
LIN {X 0,Y 83.289,Z 602.148,A -85,B 0,C 180,E1 -29112.222,E2 -29112.222} C_VEL
LIN {X 0,Y 81.705,Z 599.349,A -85,B 0,C 180,E1 -29115.359,E2 -29115.359} C_VEL
LIN {X 0,Y 80.026,Z 596.326,A -85,B 0,C 180,E1 -29119.291,E2 -29119.291} C_VEL
LIN {X 0,Y 78.143,Z 592.921,A -85,B 0,C 180,E1 -29125.244,E2 -29125.244} C_VEL
LIN {X 0,Y 76.101,Z 590.117,A -85,B 0,C 180,E1 -29138.324,E2 -29138.324} C_VEL
LIN {X 0,Y 76.3,Z 589.99,A -85,B 0,C 180,E1 -29145.49,E2 -29145.49} C_VEL
LIN {X 0,Y 78.383,Z 592.425,A -85,B 0,C 180,E1 -29156.308,E2 -29156.308} C_VEL
LIN {X 0,Y 80.257,Z 595.973,A -85,B 0,C 180,E1 -29162.031,E2 -29162.031} C_VEL
LIN {X 0,Y 82.891,Z 601.187,A -85,B 0,C 180,E1 -29167.981,E2 -29167.981} C_VEL
LIN {X 0,Y 85.793,Z 606.884,A -85,B 0,C 180,E1 -29173.075,E2 -29173.075} C_VEL
LIN {X 0,Y 88.703,Z 613.276,A -85,B 0,C 180,E1 -29177.361,E2 -29177.361} C_VEL
LIN {X 0,Y 91.107,Z 622.183,A -85,B 0,C 180,E1 -29181.046,E2 -29181.046} C_VEL
LIN {X 0,Y 93.16,Z 631.105,A -85,B 0,C 180,E1 -29184.012,E2 -29184.012} C_VEL
LIN {X 0,Y 89.646,Z 659.362,A -85,B 0,C 180,E1 -29185.719,E2 -29185.719} C_VEL
LIN {X 0,Y 86.79,Z 672.625,A -85,B 0,C 180,E1 -29187.036,E2 -29187.036} C_VEL
LIN {X 0,Y 83.131,Z 684.36,A -85,B 0,C 180,E1 -29188.707,E2 -29188.707} C_VEL
LIN {X 0,Y 78.255,Z 696.79,A -85,B 0,C 180,E1 -29191.442,E2 -29191.442} C_VEL
LIN {X 0,Y 72.885,Z 707.934,A -85,B 0,C 180,E1 -29194.961,E2 -29194.961} C_VEL
LIN {X 0,Y 67.379,Z 717.79,A -85,B 0,C 180,E1 -29199.432,E2 -29199.432} C_VEL
LIN {X 0,Y 61.054,Z 727.965,A -85,B 0,C 180,E1 -29206.319,E2 -29206.319} C_VEL
LIN {X 0,Y 55.545,Z 736.73,A -85,B 0,C 180,E1 -29215.294,E2 -29215.294} C_VEL
LIN {X 0,Y 51.58,Z 743.678,A -85,B 0,C 180,E1 -29225.874,E2 -29225.874} C_VEL
LIN {X 0,Y 49.487,Z 749.194,A -85,B 0,C 180,E1 -29237.701,E2 -29237.701} C_VEL
LIN {X 0,Y 49.377,Z 753.458,A -85,B 0,C 180,E1 -29250,E2 -29250} C_VEL
LIN {X 0,Y 49.208,Z 755.495,A -85,B 0,C 180,E1 -29258.211,E2 -29258.211} C_VEL
LIN {X 0,Y 51.323,Z 758.336,A -85,B 0,C 180,E1 -29274.255,E2 -29274.255} C_VEL
LIN {X 0,Y 57.017,Z 759.669,A -85,B 0,C 180,E1 -29288.046,E2 -29288.046} C_VEL
LIN {X 0,Y 65.579,Z 759.627,A -85,B 0,C 180,E1 -29298.604,E2 -29298.604} C_VEL
LIN {X 0,Y 75.89,Z 758.201,A -85,B 0,C 180,E1 -29306.454,E2 -29306.454} C_VEL
LIN {X 0,Y 87.353,Z 755.286,A -85,B 0,C 180,E1 -29312.249,E2 -29312.249} C_VEL
LIN {X 0,Y 99.627,Z 750.871,A -85,B 0,C 180,E1 -29316.497,E2 -29316.497} C_VEL
LIN {X 0,Y 109.197,Z 746.426,A -85,B 0,C 180,E1 -29318.941,E2 -29318.941} C_VEL
LIN {X 0,Y 120.586,Z 739.897,A -85,B 0,C 180,E1 -29321.273,E2 -29321.273} C_VEL
LIN {X 0,Y 125.549,Z 736.561,A -85,B 0,C 180,E1 -29322.102,E2 -29322.102} C_VEL
LIN {X 0,Y 124.967,Z 736.877,A -85,B 0,C 180,E1 -29322.948,E2 -29322.948} C_VEL
LIN {X 0,Y 114.316,Z 743.18,A -85,B 0,C 180,E1 -29325.198,E2 -29325.198} C_VEL
LIN {X 0,Y 102.962,Z 748.474,A -85,B 0,C 180,E1 -29328.182,E2 -29328.182} C_VEL
LIN {X 0,Y 92.311,Z 752.223,A -85,B 0,C 180,E1 -29331.777,E2 -29331.777} C_VEL
LIN {X 0,Y 90.413,Z 752.704,A -85,B 0,C 180,E1 -29332.539,E2 -29332.539} C_VEL
LIN {X 0,Y 85.268,Z 754.068,A -85,B 0,C 180,E1 -29334.272,E2 -29334.272} C_VEL
LIN {X 0,Y 76.008,Z 755.797,A -85,B 0,C 180,E1 -29336.505,E2 -29336.505} C_VEL
LIN {X 0,Y 66.837,Z 756.711,A -85,B 0,C 180,E1 -29339.385,E2 -29339.385} C_VEL
LIN {X 0,Y 61.991,Z 756.737,A -85,B 0,C 180,E1 -29342.366,E2 -29342.366} C_VEL
LIN {X 0,Y 56.704,Z 756.486,A -85,B 0,C 180,E1 -29347.468,E2 -29347.468} C_VEL
LIN {X 0,Y 50.299,Z 755.363,A -85,B 0,C 180,E1 -29356.223,E2 -29356.223} C_VEL
LIN {X 0,Y 44.993,Z 753.266,A -85,B 0,C 180,E1 -29367.939,E2 -29367.939} C_VEL
LIN {X 0,Y 41.852,Z 750.151,A -85,B 0,C 180,E1 -29382.192,E2 -29382.192} C_VEL
LIN {X 0,Y 41.548,Z 745.347,A -85,B 0,C 180,E1 -29399.506,E2 -29399.506} C_VEL
LIN {X 0,Y 43.925,Z 739.902,A -85,B 0,C 180,E1 -29413.723,E2 -29413.723} C_VEL
LIN {X 0,Y 48.635,Z 732.519,A -85,B 0,C 180,E1 -29426.884,E2 -29426.884} C_VEL
LIN {X 0,Y 55.018,Z 723.407,A -85,B 0,C 180,E1 -29437.339,E2 -29437.339} C_VEL
LIN {X 0,Y 61.821,Z 713.098,A -85,B 0,C 180,E1 -29444.82,E2 -29444.82} C_VEL
LIN {X 0,Y 67.738,Z 703.035,A -85,B 0,C 180,E1 -29449.706,E2 -29449.706} C_VEL
LIN {X 0,Y 73.234,Z 692.185,A -85,B 0,C 180,E1 -29453.301,E2 -29453.301} C_VEL
LIN {X 0,Y 78.248,Z 680.096,A -85,B 0,C 180,E1 -29456.087,E2 -29456.087} C_VEL
LIN {X 0,Y 82.454,Z 666.971,A -85,B 0,C 180,E1 -29458.162,E2 -29458.162} C_VEL
LIN {X 0,Y 85.407,Z 653.444,A -85,B 0,C 180,E1 -29459.585,E2 -29459.585} C_VEL
LIN {X 0,Y 88.96,Z 626.942,A -85,B 0,C 180,E1 -29461.088,E2 -29461.088} C_VEL
LIN {X 0,Y 86.624,Z 620.664,A -85,B 0,C 180,E1 -29464.38,E2 -29464.38} C_VEL
LIN {X 0,Y 83.244,Z 612.938,A -85,B 0,C 180,E1 -29469.799,E2 -29469.799} C_VEL
LIN {X 0,Y 80.537,Z 607.312,A -85,B 0,C 180,E1 -29475.151,E2 -29475.151} C_VEL
LIN {X 0,Y 78.208,Z 602.793,A -85,B 0,C 180,E1 -29481.024,E2 -29481.024} C_VEL
LIN {X 0,Y 76.49,Z 599.384,A -85,B 0,C 180,E1 -29487.346,E2 -29487.346} C_VEL
LIN {X 0,Y 75.028,Z 597.086,A -85,B 0,C 180,E1 -29499.503,E2 -29499.503} C_VEL
LIN {X 0,Y 75.225,Z 597.024,A -85,B 0,C 180,E1 -29505.278,E2 -29505.278} C_VEL
LIN {X 0,Y 76.888,Z 599.243,A -85,B 0,C 180,E1 -29514.928,E2 -29514.928} C_VEL
LIN {X 0,Y 78.662,Z 603.089,A -85,B 0,C 180,E1 -29521.075,E2 -29521.075} C_VEL
LIN {X 0,Y 80.842,Z 607.736,A -85,B 0,C 180,E1 -29526.435,E2 -29526.435} C_VEL
LIN {X 0,Y 83.559,Z 613.763,A -85,B 0,C 180,E1 -29531.787,E2 -29531.787} C_VEL
LIN {X 0,Y 85.335,Z 618.25,A -85,B 0,C 180,E1 -29534.784,E2 -29534.784} C_VEL
LIN {X 0,Y 87.306,Z 626.534,A -85,B 0,C 180,E1 -29538.316,E2 -29538.316} C_VEL
LIN {X 0,Y 88.583,Z 632.673,A -85,B 0,C 180,E1 -29540.541,E2 -29540.541} C_VEL
LIN {X 0,Y 85.188,Z 658.866,A -85,B 0,C 180,E1 -29542.094,E2 -29542.094} C_VEL
LIN {X 0,Y 82.287,Z 671.938,A -85,B 0,C 180,E1 -29543.348,E2 -29543.348} C_VEL
LIN {X 0,Y 78.106,Z 684.755,A -85,B 0,C 180,E1 -29545.122,E2 -29545.122} C_VEL
LIN {X 0,Y 72.637,Z 697.788,A -85,B 0,C 180,E1 -29548.009,E2 -29548.009} C_VEL
LIN {X 0,Y 66.994,Z 708.653,A -85,B 0,C 180,E1 -29551.534,E2 -29551.534} C_VEL
LIN {X 0,Y 61.019,Z 718.499,A -85,B 0,C 180,E1 -29556.271,E2 -29556.271} C_VEL
LIN {X 0,Y 54.986,Z 727.459,A -85,B 0,C 180,E1 -29562.7,E2 -29562.7} C_VEL
LIN {X 0,Y 48.975,Z 736.223,A -85,B 0,C 180,E1 -29572.42,E2 -29572.42} C_VEL
LIN {X 0,Y 44.602,Z 743.167,A -85,B 0,C 180,E1 -29584.322,E2 -29584.322} C_VEL
LIN {X 0,Y 42.261,Z 749.481,A -85,B 0,C 180,E1 -29600.427,E2 -29600.427} C_VEL
LIN {X 0,Y 42.349,Z 752.348,A -85,B 0,C 180,E1 -29610,E2 -29610} C_VEL
LIN {X 0,Y 42.247,Z 754.486,A -85,B 0,C 180,E1 -29619.576,E2 -29619.576} C_VEL
LIN {X 0,Y 44.954,Z 757.519,A -85,B 0,C 180,E1 -29637.969,E2 -29637.969} C_VEL
LIN {X 0,Y 51.608,Z 759.101,A -85,B 0,C 180,E1 -29652.913,E2 -29652.913} C_VEL
LIN {X 0,Y 61.11,Z 759.264,A -85,B 0,C 180,E1 -29663.613,E2 -29663.613} C_VEL
LIN {X 0,Y 72.203,Z 758.038,A -85,B 0,C 180,E1 -29671.165,E2 -29671.165} C_VEL
LIN {X 0,Y 84.284,Z 755.432,A -85,B 0,C 180,E1 -29676.522,E2 -29676.522} C_VEL
LIN {X 0,Y 97.022,Z 751.263,A -85,B 0,C 180,E1 -29680.332,E2 -29680.332} C_VEL
LIN {X 0,Y 104.753,Z 748.048,A -85,B 0,C 180,E1 -29682.045,E2 -29682.045} C_VEL
LIN {X 0,Y 106.812,Z 747.032,A -85,B 0,C 180,E1 -29682.975,E2 -29682.975} C_VEL
LIN {X 0,Y 94.054,Z 751.804,A -85,B 0,C 180,E1 -29686.257,E2 -29686.257} C_VEL
LIN {X 0,Y 82.77,Z 754.707,A -85,B 0,C 180,E1 -29690.22,E2 -29690.22} C_VEL
LIN {X 0,Y 70.423,Z 756.517,A -85,B 0,C 180,E1 -29696.322,E2 -29696.322} C_VEL
LIN {X 0,Y 61.991,Z 756.737,A -85,B 0,C 180,E1 -29702.366,E2 -29702.366} C_VEL
LIN {X 0,Y 57.326,Z 756.612,A -85,B 0,C 180,E1 -29705.849,E2 -29705.849} C_VEL
LIN {X 0,Y 48.916,Z 755.756,A -85,B 0,C 180,E1 -29711.477,E2 -29711.477} C_VEL
LIN {X 0,Y 42.555,Z 754.529,A -85,B 0,C 180,E1 -29717.302,E2 -29717.302} C_VEL
LIN {X 0,Y 38.783,Z 753.237,A -85,B 0,C 180,E1 -29723.498,E2 -29723.498} C_VEL
LIN {X 0,Y 37.865,Z 752.724,A -85,B 0,C 180,E1 -29726.01,E2 -29726.01} C_VEL
LIN {X 0,Y 34.473,Z 748.926,A -85,B 0,C 180,E1 -29744.478,E2 -29744.478} C_VEL
LIN {X 0,Y 34.545,Z 744.832,A -85,B 0,C 180,E1 -29760.953,E2 -29760.953} C_VEL
LIN {X 0,Y 37.864,Z 738.509,A -85,B 0,C 180,E1 -29779.304,E2 -29779.304} C_VEL
LIN {X 0,Y 43.187,Z 731.285,A -85,B 0,C 180,E1 -29792.644,E2 -29792.644} C_VEL
LIN {X 0,Y 49.963,Z 722.347,A -85,B 0,C 180,E1 -29802.806,E2 -29802.806} C_VEL
LIN {X 0,Y 57.023,Z 712.419,A -85,B 0,C 180,E1 -29809.811,E2 -29809.811} C_VEL
LIN {X 0,Y 63.708,Z 701.492,A -85,B 0,C 180,E1 -29814.766,E2 -29814.766} C_VEL
LIN {X 0,Y 70.09,Z 689.054,A -85,B 0,C 180,E1 -29818.442,E2 -29818.442} C_VEL
LIN {X 0,Y 74.781,Z 677.578,A -85,B 0,C 180,E1 -29820.731,E2 -29820.731} C_VEL
LIN {X 0,Y 78.969,Z 664.087,A -85,B 0,C 180,E1 -29822.54,E2 -29822.54} C_VEL
LIN {X 0,Y 81.733,Z 650.934,A -85,B 0,C 180,E1 -29823.721,E2 -29823.721} C_VEL
LIN {X 0,Y 84.613,Z 629.368,A -85,B 0,C 180,E1 -29824.865,E2 -29824.865} C_VEL
LIN {X 0,Y 83.025,Z 624.769,A -85,B 0,C 180,E1 -29827.551,E2 -29827.551} C_VEL
LIN {X 0,Y 80.082,Z 617.264,A -85,B 0,C 180,E1 -29833.303,E2 -29833.303} C_VEL
LIN {X 0,Y 77.663,Z 611.957,A -85,B 0,C 180,E1 -29839.055,E2 -29839.055} C_VEL
LIN {X 0,Y 76.368,Z 609.107,A -85,B 0,C 180,E1 -29843.159,E2 -29843.159} C_VEL
LIN {X 0,Y 75.007,Z 606.092,A -85,B 0,C 180,E1 -29849.033,E2 -29849.033} C_VEL
LIN {X 0,Y 73.972,Z 604.101,A -85,B 0,C 180,E1 -29859.718,E2 -29859.718} C_VEL
LIN {X 0,Y 74.151,Z 604.043,A -85,B 0,C 180,E1 -29865.06,E2 -29865.06} C_VEL
LIN {X 0,Y 75.423,Z 605.94,A -85,B 0,C 180,E1 -29873.368,E2 -29873.368} C_VEL
LIN {X 0,Y 76.817,Z 609.496,A -85,B 0,C 180,E1 -29879.17,E2 -29879.17} C_VEL
LIN {X 0,Y 78.866,Z 614.322,A -85,B 0,C 180,E1 -29884.897,E2 -29884.897} C_VEL
LIN {X 0,Y 81.214,Z 620.409,A -85,B 0,C 180,E1 -29890.162,E2 -29890.162} C_VEL
LIN {X 0,Y 82.142,Z 623.308,A -85,B 0,C 180,E1 -29892.045,E2 -29892.045} C_VEL
LIN {X 0,Y 84.11,Z 633.175,A -85,B 0,C 180,E1 -29896.292,E2 -29896.292} C_VEL
LIN {X 0,Y 84.35,Z 634.441,A -85,B 0,C 180,E1 -29896.776,E2 -29896.776} C_VEL
LIN {X 0,Y 80.907,Z 659.323,A -85,B 0,C 180,E1 -29898.192,E2 -29898.192} C_VEL
LIN {X 0,Y 77.963,Z 671.79,A -85,B 0,C 180,E1 -29899.319,E2 -29899.319} C_VEL
LIN {X 0,Y 73.814,Z 684.017,A -85,B 0,C 180,E1 -29900.893,E2 -29900.893} C_VEL
LIN {X 0,Y 68.825,Z 695.526,A -85,B 0,C 180,E1 -29903.219,E2 -29903.219} C_VEL
LIN {X 0,Y 62.605,Z 707.128,A -85,B 0,C 180,E1 -29906.686,E2 -29906.686} C_VEL
LIN {X 0,Y 56.418,Z 716.871,A -85,B 0,C 180,E1 -29911.086,E2 -29911.086} C_VEL
LIN {X 0,Y 49.208,Z 726.841,A -85,B 0,C 180,E1 -29918.233,E2 -29918.233} C_VEL
LIN {X 0,Y 42.568,Z 735.638,A -85,B 0,C 180,E1 -29928.671,E2 -29928.671} C_VEL
LIN {X 0,Y 37.681,Z 742.619,A -85,B 0,C 180,E1 -29942.208,E2 -29942.208} C_VEL
LIN {X 0,Y 35.298,Z 748.157,A -85,B 0,C 180,E1 -29958.516,E2 -29958.516} C_VEL
LIN {X 0,Y 35.301,Z 751.145,A -85,B 0,C 180,E1 -29970,E2 -29970} C_VEL
LIN {X 0,Y 35.324,Z 753.446,A -85,B 0,C 180,E1 -29981.476,E2 -29981.476} C_VEL
LIN {X 0,Y 38.839,Z 756.674,A -85,B 0,C 180,E1 -30002.877,E2 -30002.877} C_VEL
LIN {X 0,Y 46.658,Z 758.449,A -85,B 0,C 180,E1 -30018.861,E2 -30018.861} C_VEL
LIN {X 0,Y 57.179,Z 758.875,A -85,B 0,C 180,E1 -30029.358,E2 -30029.358} C_VEL
LIN {X 0,Y 69.053,Z 757.887,A -85,B 0,C 180,E1 -30036.343,E2 -30036.343} C_VEL
LIN {X 0,Y 81.712,Z 755.494,A -85,B 0,C 180,E1 -30041.099,E2 -30041.099} C_VEL
LIN {X 0,Y 88.248,Z 753.758,A -85,B 0,C 180,E1 -30042.871,E2 -30042.871} C_VEL
LIN {X 0,Y 88.126,Z 753.768,A -85,B 0,C 180,E1 -30043.132,E2 -30043.132} C_VEL
LIN {X 0,Y 79.771,Z 755.567,A -85,B 0,C 180,E1 -30045.72,E2 -30045.72} C_VEL
LIN {X 0,Y 71.612,Z 756.694,A -85,B 0,C 180,E1 -30048.927,E2 -30048.927} C_VEL
LIN {X 0,Y 62.722,Z 757.248,A -85,B 0,C 180,E1 -30053.563,E2 -30053.563} C_VEL
LIN {X 0,Y 54.018,Z 756.982,A -85,B 0,C 180,E1 -30059.996,E2 -30059.996} C_VEL
LIN {X 0,Y 46.199,Z 755.82,A -85,B 0,C 180,E1 -30068.746,E2 -30068.746} C_VEL
LIN {X 0,Y 37.865,Z 752.724,A -85,B 0,C 180,E1 -30086.01,E2 -30086.01} C_VEL
LIN {X 0,Y 35.181,Z 751.099,A -85,B 0,C 180,E1 -30093.864,E2 -30093.864} C_VEL
LIN {X 0,Y 30.626,Z 747.778,A -85,B 0,C 180,E1 -30108.19,E2 -30108.19} C_VEL
LIN {X 0,Y 28.361,Z 743.734,A -85,B 0,C 180,E1 -30125.428,E2 -30125.428} C_VEL
LIN {X 0,Y 29.31,Z 740.934,A -85,B 0,C 180,E1 -30135.689,E2 -30135.689} C_VEL
LIN {X 0,Y 34.499,Z 734.301,A -85,B 0,C 180,E1 -30152.541,E2 -30152.541} C_VEL
LIN {X 0,Y 41.463,Z 726.084,A -85,B 0,C 180,E1 -30164.734,E2 -30164.734} C_VEL
LIN {X 0,Y 49.351,Z 716.276,A -85,B 0,C 180,E1 -30173.055,E2 -30173.055} C_VEL
LIN {X 0,Y 56.678,Z 705.707,A -85,B 0,C 180,E1 -30178.419,E2 -30178.419} C_VEL
LIN {X 0,Y 63.078,Z 694.79,A -85,B 0,C 180,E1 -30181.953,E2 -30181.953} C_VEL
LIN {X 0,Y 68.894,Z 682.506,A -85,B 0,C 180,E1 -30184.578,E2 -30184.578} C_VEL
LIN {X 0,Y 73.632,Z 669.487,A -85,B 0,C 180,E1 -30186.421,E2 -30186.421} C_VEL
LIN {X 0,Y 76.955,Z 656.597,A -85,B 0,C 180,E1 -30187.672,E2 -30187.672} C_VEL
LIN {X 0,Y 79.682,Z 639.546,A -85,B 0,C 180,E1 -30188.57,E2 -30188.57} C_VEL
LIN {X 0,Y 80.657,Z 631.715,A -85,B 0,C 180,E1 -30189.031,E2 -30189.031} C_VEL
LIN {X 0,Y 77.991,Z 624.05,A -85,B 0,C 180,E1 -30194.852,E2 -30194.852} C_VEL
LIN {X 0,Y 75.921,Z 618.571,A -85,B 0,C 180,E1 -30200.584,E2 -30200.584} C_VEL
LIN {X 0,Y 74.649,Z 615.418,A -85,B 0,C 180,E1 -30205.362,E2 -30205.362} C_VEL
LIN {X 0,Y 73.667,Z 612.933,A -85,B 0,C 180,E1 -30210.333,E2 -30210.333} C_VEL
LIN {X 0,Y 72.911,Z 611.081,A -85,B 0,C 180,E1 -30220.654,E2 -30220.654} C_VEL
LIN {X 0,Y 73.077,Z 611.071,A -85,B 0,C 180,E1 -30224.834,E2 -30224.834} C_VEL
LIN {X 0,Y 74.023,Z 612.773,A -85,B 0,C 180,E1 -30231.994,E2 -30231.994} C_VEL
LIN {X 0,Y 75.088,Z 615.926,A -85,B 0,C 180,E1 -30237.264,E2 -30237.264} C_VEL
LIN {X 0,Y 76.688,Z 620.408,A -85,B 0,C 180,E1 -30242.669,E2 -30242.669} C_VEL
LIN {X 0,Y 78.917,Z 626.971,A -85,B 0,C 180,E1 -30248.391,E2 -30248.391} C_VEL
LIN {X 0,Y 80.409,Z 636.333,A -85,B 0,C 180,E1 -30252.669,E2 -30252.669} C_VEL
LIN {X 0,Y 77.129,Z 658.904,A -85,B 0,C 180,E1 -30253.85,E2 -30253.85} C_VEL
LIN {X 0,Y 73.949,Z 671.788,A -85,B 0,C 180,E1 -30254.892,E2 -30254.892} C_VEL
LIN {X 0,Y 69.573,Z 684.092,A -85,B 0,C 180,E1 -30256.334,E2 -30256.334} C_VEL
LIN {X 0,Y 63.967,Z 696.277,A -85,B 0,C 180,E1 -30258.63,E2 -30258.63} C_VEL
LIN {X 0,Y 57.371,Z 707.779,A -85,B 0,C 180,E1 -30261.93,E2 -30261.93} C_VEL
LIN {X 0,Y 50.896,Z 717.206,A -85,B 0,C 180,E1 -30266.163,E2 -30266.163} C_VEL
LIN {X 0,Y 43.801,Z 726.219,A -85,B 0,C 180,E1 -30272.61,E2 -30272.61} C_VEL
LIN {X 0,Y 36.395,Z 735.044,A -85,B 0,C 180,E1 -30283.604,E2 -30283.604} C_VEL
LIN {X 0,Y 30.832,Z 742.063,A -85,B 0,C 180,E1 -30299.145,E2 -30299.145} C_VEL
LIN {X 0,Y 28.384,Z 746.777,A -85,B 0,C 180,E1 -30315.665,E2 -30315.665} C_VEL
LIN {X 0,Y 28.244,Z 749.903,A -85,B 0,C 180,E1 -30330,E2 -30330} C_VEL
LIN {X 0,Y 28.323,Z 751.168,A -85,B 0,C 180,E1 -30336.937,E2 -30336.937} C_VEL
LIN {X 0,Y 30.058,Z 754.231,A -85,B 0,C 180,E1 -30357.88,E2 -30357.88} C_VEL
LIN {X 0,Y 37.308,Z 756.977,A -85,B 0,C 180,E1 -30378.894,E2 -30378.894} C_VEL
LIN {X 0,Y 47.964,Z 758.274,A -85,B 0,C 180,E1 -30391.538,E2 -30391.538} C_VEL
LIN {X 0,Y 60.115,Z 758.215,A -85,B 0,C 180,E1 -30399.268,E2 -30399.268} C_VEL
LIN {X 0,Y 66.514,Z 757.682,A -85,B 0,C 180,E1 -30401.978,E2 -30401.978} C_VEL
LIN {X 0,Y 67.975,Z 757.428,A -85,B 0,C 180,E1 -30403.936,E2 -30403.936} C_VEL
LIN {X 0,Y 57.314,Z 757.706,A -85,B 0,C 180,E1 -30408.801,E2 -30408.801} C_VEL
LIN {X 0,Y 49.47,Z 757.19,A -85,B 0,C 180,E1 -30413.955,E2 -30413.955} C_VEL
LIN {X 0,Y 42.173,Z 756.103,A -85,B 0,C 180,E1 -30420.973,E2 -30420.973} C_VEL
LIN {X 0,Y 32.775,Z 753.145,A -85,B 0,C 180,E1 -30437.197,E2 -30437.197} C_VEL
LIN {X 0,Y 27.657,Z 748.965,A -85,B 0,C 180,E1 -30460.331,E2 -30460.331} C_VEL
LIN {X 0,Y 28.029,Z 743.148,A -85,B 0,C 180,E1 -30487.707,E2 -30487.707} C_VEL
LIN {X 0,Y 29.31,Z 740.934,A -85,B 0,C 180,E1 -30495.689,E2 -30495.689} C_VEL
LIN {X 0,Y 30.454,Z 738.963,A -85,B 0,C 180,E1 -30501.78,E2 -30501.78} C_VEL
LIN {X 0,Y 31.79,Z 735.82,A -85,B 0,C 180,E1 -30510.646,E2 -30510.646} C_VEL
LIN {X 0,Y 35.693,Z 727.61,A -85,B 0,C 180,E1 -30528.782,E2 -30528.782} C_VEL
LIN {X 0,Y 38.549,Z 723.661,A -85,B 0,C 180,E1 -30534.186,E2 -30534.186} C_VEL
LIN {X 0,Y 39.712,Z 722.278,A -85,B 0,C 180,E1 -30535.501,E2 -30535.501} C_VEL
LIN {X 0,Y 47.24,Z 713.176,A -85,B 0,C 180,E1 -30541.384,E2 -30541.384} C_VEL
LIN {X 0,Y 54.504,Z 702.801,A -85,B 0,C 180,E1 -30545.467,E2 -30545.467} C_VEL
LIN {X 0,Y 61.118,Z 691.383,A -85,B 0,C 180,E1 -30548.287,E2 -30548.287} C_VEL
LIN {X 0,Y 66.427,Z 679.97,A -85,B 0,C 180,E1 -30550.179,E2 -30550.179} C_VEL
LIN {X 0,Y 71.01,Z 666.957,A -85,B 0,C 180,E1 -30551.632,E2 -30551.632} C_VEL
LIN {X 0,Y 74.258,Z 653.639,A -85,B 0,C 180,E1 -30552.622,E2 -30552.622} C_VEL
LIN {X 0,Y 77.117,Z 634.82,A -85,B 0,C 180,E1 -30553.405,E2 -30553.405} C_VEL
LIN {X 0,Y 75.227,Z 628.443,A -85,B 0,C 180,E1 -30558.679,E2 -30558.679} C_VEL
LIN {X 0,Y 73.74,Z 623.935,A -85,B 0,C 180,E1 -30564.114,E2 -30564.114} C_VEL
LIN {X 0,Y 72.951,Z 621.626,A -85,B 0,C 180,E1 -30567.826,E2 -30567.826} C_VEL
LIN {X 0,Y 72.36,Z 619.736,A -85,B 0,C 180,E1 -30571.743,E2 -30571.743} C_VEL
LIN {X 0,Y 71.86,Z 618.12,A -85,B 0,C 180,E1 -30580.36,E2 -30580.36} C_VEL
LIN {X 0,Y 72.007,Z 618.196,A -85,B 0,C 180,E1 -30584.818,E2 -30584.818} C_VEL
LIN {X 0,Y 72.677,Z 619.692,A -85,B 0,C 180,E1 -30590.748,E2 -30590.748} C_VEL
LIN {X 0,Y 73.483,Z 622.538,A -85,B 0,C 180,E1 -30595.488,E2 -30595.488} C_VEL
LIN {X 0,Y 74.821,Z 627.232,A -85,B 0,C 180,E1 -30601.014,E2 -30601.014} C_VEL
LIN {X 0,Y 76.089,Z 631.589,A -85,B 0,C 180,E1 -30604.934,E2 -30604.934} C_VEL
LIN {X 0,Y 76.918,Z 638.108,A -85,B 0,C 180,E1 -30608.132,E2 -30608.132} C_VEL
LIN {X 0,Y 73.808,Z 658.624,A -85,B 0,C 180,E1 -30609.097,E2 -30609.097} C_VEL
LIN {X 0,Y 70.673,Z 670.966,A -85,B 0,C 180,E1 -30609.933,E2 -30609.933} C_VEL
LIN {X 0,Y 66.241,Z 683.183,A -85,B 0,C 180,E1 -30611.073,E2 -30611.073} C_VEL
LIN {X 0,Y 60.414,Z 695.468,A -85,B 0,C 180,E1 -30613.031,E2 -30613.031} C_VEL
LIN {X 0,Y 53.256,Z 707.367,A -85,B 0,C 180,E1 -30615.945,E2 -30615.945} C_VEL
LIN {X 0,Y 46.611,Z 716.482,A -85,B 0,C 180,E1 -30619.551,E2 -30619.551} C_VEL
LIN {X 0,Y 38.932,Z 725.519,A -85,B 0,C 180,E1 -30625.501,E2 -30625.501} C_VEL
LIN {X 0,Y 30.633,Z 734.365,A -85,B 0,C 180,E1 -30636.586,E2 -30636.586} C_VEL
LIN {X 0,Y 24.145,Z 741.434,A -85,B 0,C 180,E1 -30654.399,E2 -30654.399} C_VEL
LIN {X 0,Y 21.123,Z 748.044,A -85,B 0,C 180,E1 -30686.678,E2 -30686.678} C_VEL
LIN {X 0,Y 21.393,Z 749.974,A -85,B 0,C 180,E1 -30699.697,E2 -30699.697} C_VEL
LIN {X 0,Y 24.048,Z 753.18,A -85,B 0,C 180,E1 -30725.766,E2 -30725.766} C_VEL
LIN {X 0,Y 33.092,Z 756.116,A -85,B 0,C 180,E1 -30748.156,E2 -30748.156} C_VEL
LIN {X 0,Y 45.017,Z 757.693,A -85,B 0,C 180,E1 -30759.503,E2 -30759.503} C_VEL
LIN {X 0,Y 51.409,Z 757.951,A -85,B 0,C 180,E1 -30763.122,E2 -30763.122} C_VEL
LIN {X 0,Y 51.28,Z 757.92,A -85,B 0,C 180,E1 -30763.605,E2 -30763.605} C_VEL
LIN {X 0,Y 40.938,Z 756.697,A -85,B 0,C 180,E1 -30770.11,E2 -30770.11} C_VEL
LIN {X 0,Y 31.879,Z 754.607,A -85,B 0,C 180,E1 -30779.994,E2 -30779.994} C_VEL
LIN {X 0,Y 22.861,Z 750.599,A -85,B 0,C 180,E1 -30802.741,E2 -30802.741} C_VEL
LIN {X 0,Y 20.122,Z 745.129,A -85,B 0,C 180,E1 -30838.406,E2 -30838.406} C_VEL
LIN {X 0,Y 23.188,Z 739.927,A -85,B 0,C 180,E1 -30863.477,E2 -30863.477} C_VEL
LIN {X 0,Y 28.507,Z 734.185,A -85,B 0,C 180,E1 -30879.588,E2 -30879.588} C_VEL
LIN {X 0,Y 36.774,Z 725.544,A -85,B 0,C 180,E1 -30892.471,E2 -30892.471} C_VEL
LIN {X 0,Y 39.712,Z 722.278,A -85,B 0,C 180,E1 -30895.501,E2 -30895.501} C_VEL
LIN {X 0,Y 42.885,Z 718.123,A -85,B 0,C 180,E1 -30899.345,E2 -30899.345} C_VEL
LIN {X 0,Y 47.09,Z 710.873,A -85,B 0,C 180,E1 -30906.148,E2 -30906.148} C_VEL
LIN {X 0,Y 51.262,Z 703.117,A -85,B 0,C 180,E1 -30911.555,E2 -30911.555} C_VEL
LIN {X 0,Y 54.127,Z 698.166,A -85,B 0,C 180,E1 -30913.254,E2 -30913.254} C_VEL
LIN {X 0,Y 60.702,Z 686.08,A -85,B 0,C 180,E1 -30915.164,E2 -30915.164} C_VEL
LIN {X 0,Y 66.003,Z 673.414,A -85,B 0,C 180,E1 -30916.501,E2 -30916.501} C_VEL
LIN {X 0,Y 70.144,Z 659.617,A -85,B 0,C 180,E1 -30917.442,E2 -30917.442} C_VEL
LIN {X 0,Y 72.759,Z 645.965,A -85,B 0,C 180,E1 -30918.008,E2 -30918.008} C_VEL
LIN {X 0,Y 73.933,Z 637.749,A -85,B 0,C 180,E1 -30918.29,E2 -30918.29} C_VEL
LIN {X 0,Y 72.642,Z 632.279,A -85,B 0,C 180,E1 -30923.545,E2 -30923.545} C_VEL
LIN {X 0,Y 71.507,Z 628.181,A -85,B 0,C 180,E1 -30929.632,E2 -30929.632} C_VEL
LIN {X 0,Y 71.056,Z 626.458,A -85,B 0,C 180,E1 -30933.601,E2 -30933.601} C_VEL
LIN {X 0,Y 70.806,Z 625.203,A -85,B 0,C 180,E1 -30940.055,E2 -30940.055} C_VEL
LIN {X 0,Y 70.908,Z 625.167,A -85,B 0,C 180,E1 -30944.111,E2 -30944.111} C_VEL
LIN {X 0,Y 71.35,Z 626.423,A -85,B 0,C 180,E1 -30949.207,E2 -30949.207} C_VEL
LIN {X 0,Y 71.994,Z 629.314,A -85,B 0,C 180,E1 -30953.895,E2 -30953.895} C_VEL
LIN {X 0,Y 73.034,Z 634.022,A -85,B 0,C 180,E1 -30959.302,E2 -30959.302} C_VEL
LIN {X 0,Y 73.586,Z 637.034,A -85,B 0,C 180,E1 -30961.716,E2 -30961.716} C_VEL
LIN {X 0,Y 73.843,Z 640.012,A -85,B 0,C 180,E1 -30963.248,E2 -30963.248} C_VEL
LIN {X 0,Y 70.888,Z 658.572,A -85,B 0,C 180,E1 -30963.979,E2 -30963.979} C_VEL
LIN {X 0,Y 67.58,Z 671.056,A -85,B 0,C 180,E1 -30964.613,E2 -30964.613} C_VEL
LIN {X 0,Y 62.664,Z 683.933,A -85,B 0,C 180,E1 -30965.533,E2 -30965.533} C_VEL
LIN {X 0,Y 56.649,Z 695.974,A -85,B 0,C 180,E1 -30967.035,E2 -30967.035} C_VEL
LIN {X 0,Y 49.817,Z 706.812,A -85,B 0,C 180,E1 -30969.067,E2 -30969.067} C_VEL
LIN {X 0,Y 41.403,Z 717.603,A -85,B 0,C 180,E1 -30972.571,E2 -30972.571} C_VEL
LIN {X 0,Y 33.229,Z 726.396,A -85,B 0,C 180,E1 -30977.874,E2 -30977.874} C_VEL
LIN {X 0,Y 24.078,Z 734.981,A -85,B 0,C 180,E1 -30988.88,E2 -30988.88} C_VEL
LIN {X 0,Y 16.702,Z 741.794,A -85,B 0,C 180,E1 -31010.863,E2 -31010.863} C_VEL
LIN {X 0,Y 14.148,Z 747.209,A -85,B 0,C 180,E1 -31050,E2 -31050} C_VEL
LIN {X 0,Y 14.577,Z 748.793,A -85,B 0,C 180,E1 -31065.309,E2 -31065.309} C_VEL
LIN {X 0,Y 18.784,Z 752.058,A -85,B 0,C 180,E1 -31098.44,E2 -31098.44} C_VEL
LIN {X 0,Y 29.97,Z 755.241,A -85,B 0,C 180,E1 -31119.713,E2 -31119.713} C_VEL
LIN {X 0,Y 32.52,Z 755.615,A -85,B 0,C 180,E1 -31124.462,E2 -31124.462} C_VEL
LIN {X 0,Y 20.768,Z 751.987,A -85,B 0,C 180,E1 -31139.99,E2 -31139.99} C_VEL
LIN {X 0,Y 13.899,Z 747.819,A -85,B 0,C 180,E1 -31170.359,E2 -31170.359} C_VEL
LIN {X 0,Y 14.354,Z 742.338,A -85,B 0,C 180,E1 -31218.227,E2 -31218.227} C_VEL
LIN {X 0,Y 20.627,Z 736.284,A -85,B 0,C 180,E1 -31244.815,E2 -31244.815} C_VEL
LIN {X 0,Y 29.221,Z 728.532,A -85,B 0,C 180,E1 -31258.751,E2 -31258.751} C_VEL
LIN {X 0,Y 37.602,Z 720.061,A -85,B 0,C 180,E1 -31265.737,E2 -31265.737} C_VEL
LIN {X 0,Y 46.546,Z 709.338,A -85,B 0,C 180,E1 -31270.448,E2 -31270.448} C_VEL
LIN {X 0,Y 54.127,Z 698.166,A -85,B 0,C 180,E1 -31273.254,E2 -31273.254} C_VEL
LIN {X 0,Y 56.772,Z 693.217,A -85,B 0,C 180,E1 -31274.727,E2 -31274.727} C_VEL
LIN {X 0,Y 60.104,Z 684.779,A -85,B 0,C 180,E1 -31278.405,E2 -31278.405} C_VEL
LIN {X 0,Y 63.05,Z 675.817,A -85,B 0,C 180,E1 -31281.662,E2 -31281.662} C_VEL
LIN {X 0,Y 64.903,Z 670.147,A -85,B 0,C 180,E1 -31282.583,E2 -31282.583} C_VEL
LIN {X 0,Y 68.483,Z 657.313,A -85,B 0,C 180,E1 -31283.126,E2 -31283.126} C_VEL
LIN {X 0,Y 71.318,Z 640.843,A -85,B 0,C 180,E1 -31283.539,E2 -31283.539} C_VEL
LIN {X 0,Y 70.493,Z 636.581,A -85,B 0,C 180,E1 -31288.506,E2 -31288.506} C_VEL
LIN {X 0,Y 69.959,Z 633.688,A -85,B 0,C 180,E1 -31293.673,E2 -31293.673} C_VEL
LIN {X 0,Y 69.758,Z 632.146,A -85,B 0,C 180,E1 -31301.082,E2 -31301.082} C_VEL
LIN {X 0,Y 69.853,Z 632.314,A -85,B 0,C 180,E1 -31304.338,E2 -31304.338} C_VEL
LIN {X 0,Y 70.09,Z 633.26,A -85,B 0,C 180,E1 -31307.805,E2 -31307.805} C_VEL
LIN {X 0,Y 70.617,Z 636.697,A -85,B 0,C 180,E1 -31312.953,E2 -31312.953} C_VEL
LIN {X 0,Y 71.268,Z 641.104,A -85,B 0,C 180,E1 -31317.502,E2 -31317.502} C_VEL
LIN {X 0,Y 71.304,Z 642.076,A -85,B 0,C 180,E1 -31318.036,E2 -31318.036} C_VEL
LIN {X 0,Y 68.368,Z 659.409,A -85,B 0,C 180,E1 -31318.53,E2 -31318.53} C_VEL
LIN {X 0,Y 64.687,Z 672.404,A -85,B 0,C 180,E1 -31318.933,E2 -31318.933} C_VEL
LIN {X 0,Y 59.74,Z 684.674,A -85,B 0,C 180,E1 -31319.404,E2 -31319.404} C_VEL
LIN {X 0,Y 53.583,Z 696.464,A -85,B 0,C 180,E1 -31320.229,E2 -31320.229} C_VEL
LIN {X 0,Y 46.574,Z 707.102,A -85,B 0,C 180,E1 -31321.425,E2 -31321.425} C_VEL
LIN {X 0,Y 38.715,Z 716.796,A -85,B 0,C 180,E1 -31323.251,E2 -31323.251} C_VEL
LIN {X 0,Y 30.057,Z 725.622,A -85,B 0,C 180,E1 -31326.422,E2 -31326.422} C_VEL
LIN {X 0,Y 19.915,Z 734.26,A -85,B 0,C 180,E1 -31333.958,E2 -31333.958} C_VEL
LIN {X 0,Y 10.692,Z 741.104,A -85,B 0,C 180,E1 -31354.751,E2 -31354.751} C_VEL
LIN {X 0,Y 7.075,Z 745.748,A -85,B 0,C 180,E1 -31410,E2 -31410} C_VEL
LIN {X 0,Y 8.154,Z 747.505,A -85,B 0,C 180,E1 -31440.421,E2 -31440.421} C_VEL
LIN {X 0,Y 15.067,Z 750.856,A -85,B 0,C 180,E1 -31478.891,E2 -31478.891} C_VEL
LIN {X 0,Y 14.527,Z 750.557,A -85,B 0,C 180,E1 -31485.358,E2 -31485.358} C_VEL
LIN {X 0,Y 5.88,Z 744.815,A -85,B 0,C 180,E1 -31552.732,E2 -31552.732} C_VEL
LIN {X 0,Y 12.486,Z 738.637,A -85,B 0,C 180,E1 -31614.97,E2 -31614.97} C_VEL
LIN {X 0,Y 22.305,Z 731.222,A -85,B 0,C 180,E1 -31629.061,E2 -31629.061} C_VEL
LIN {X 0,Y 32.283,Z 722.297,A -85,B 0,C 180,E1 -31635.033,E2 -31635.033} C_VEL
LIN {X 0,Y 41.776,Z 711.869,A -85,B 0,C 180,E1 -31638.209,E2 -31638.209} C_VEL
LIN {X 0,Y 50.297,Z 700.263,A -85,B 0,C 180,E1 -31640.219,E2 -31640.219} C_VEL
LIN {X 0,Y 56.787,Z 689.172,A -85,B 0,C 180,E1 -31641.368,E2 -31641.368} C_VEL
LIN {X 0,Y 62.659,Z 676.281,A -85,B 0,C 180,E1 -31642.272,E2 -31642.272} C_VEL
LIN {X 0,Y 64.903,Z 670.147,A -85,B 0,C 180,E1 -31642.583,E2 -31642.583} C_VEL
LIN {X 0,Y 65.94,Z 666.401,A -85,B 0,C 180,E1 -31643.338,E2 -31643.338} C_VEL
LIN {X 0,Y 66.874,Z 660.43,A -85,B 0,C 180,E1 -31645.93,E2 -31645.93} C_VEL
LIN {X 0,Y 67.614,Z 654.372,A -85,B 0,C 180,E1 -31648.425,E2 -31648.425} C_VEL
LIN {X 0,Y 68.193,Z 650.485,A -85,B 0,C 180,E1 -31649.042,E2 -31649.042} C_VEL
LIN {X 0,Y 69.181,Z 644.295,A -85,B 0,C 180,E1 -31649.083,E2 -31649.083} C_VEL
LIN {X 0,Y 68.812,Z 641.151,A -85,B 0,C 180,E1 -31653.869,E2 -31653.869} C_VEL
LIN {X 0,Y 68.746,Z 640.208,A -85,B 0,C 180,E1 -31655.866,E2 -31655.866} C_VEL
LIN {X 0,Y 68.73,Z 639.109,A -85,B 0,C 180,E1 -31662.139,E2 -31662.139} C_VEL
LIN {X 0,Y 68.865,Z 640.04,A -85,B 0,C 180,E1 -31666.214,E2 -31666.214} C_VEL
LIN {X 0,Y 69.117,Z 643.498,A -85,B 0,C 180,E1 -31670.999,E2 -31670.999} C_VEL
LIN {X 0,Y 69.255,Z 644.771,A -85,B 0,C 180,E1 -31672.446,E2 -31672.446} C_VEL
LIN {X 0,Y 66.551,Z 659.842,A -85,B 0,C 180,E1 -31672.674,E2 -31672.674} C_VEL
LIN {X 0,Y 62.873,Z 672.402,A -85,B 0,C 180,E1 -31672.76,E2 -31672.76} C_VEL
LIN {X 0,Y 57.568,Z 685.247,A -85,B 0,C 180,E1 -31672.699,E2 -31672.699} C_VEL
LIN {X 0,Y 51.357,Z 696.802,A -85,B 0,C 180,E1 -31672.764,E2 -31672.764} C_VEL
LIN {X 0,Y 44.268,Z 707.242,A -85,B 0,C 180,E1 -31672.852,E2 -31672.852} C_VEL
LIN {X 0,Y 35.408,Z 717.774,A -85,B 0,C 180,E1 -31672.941,E2 -31672.941} C_VEL
LIN {X 0,Y 26.552,Z 726.349,A -85,B 0,C 180,E1 -31673.009,E2 -31673.009} C_VEL
LIN {X 0,Y 17.686,Z 733.461,A -85,B 0,C 180,E1 -31673.433,E2 -31673.433} C_VEL
LIN {X 0,Y 7.067,Z 740.395,A -85,B 0,C 180,E1 -31673.963,E2 -31673.963} C_VEL
LIN {X 0,Y 5.983,Z 740.999,A -85,B 0,C 180,E1 -31674.023,E2 -31674.023} C_VEL
LIN {X 0,Y 4.055,Z 741.954,A -85,B 0,C 180,E1 -31658.839,E2 -31658.839} C_VEL
LIN {X 0,Y 15.005,Z 735.009,A -85,B 0,C 180,E1 -31647.909,E2 -31647.909} C_VEL
LIN {X 0,Y 24.974,Z 727.206,A -85,B 0,C 180,E1 -31647.586,E2 -31647.586} C_VEL
LIN {X 0,Y 35.017,Z 717.533,A -85,B 0,C 180,E1 -31647.757,E2 -31647.757} C_VEL
LIN {X 0,Y 43.467,Z 707.457,A -85,B 0,C 180,E1 -31648.085,E2 -31648.085} C_VEL
LIN {X 0,Y 50.785,Z 696.77,A -85,B 0,C 180,E1 -31648.275,E2 -31648.275} C_VEL
LIN {X 0,Y 56.99,Z 685.47,A -85,B 0,C 180,E1 -31648.498,E2 -31648.498} C_VEL
LIN {X 0,Y 62.61,Z 671.941,A -85,B 0,C 180,E1 -31648.728,E2 -31648.728} C_VEL
LIN {X 0,Y 66.49,Z 658.879,A -85,B 0,C 180,E1 -31648.949,E2 -31648.949} C_VEL
LIN {X 0,Y 68.193,Z 650.485,A -85,B 0,C 180,E1 -31649.042,E2 -31649.042} C_VEL
LIN {X 0,Y 68.404,Z 648.457,A -85,B 0,C 180,E1 -31649.7,E2 -31649.7} C_VEL
LIN {X 0,Y 68.343,Z 646.59,A -85,B 0,C 180,E1 -31651.556,E2 -31651.556} C_VEL
LIN {X 0,Y 68.16,Z 645.445,A -85,B 0,C 180,E1 -31653.97,E2 -31653.97} C_VEL
LIN {X 0,Y 67.884,Z 644.984,A -85,B 0,C 180,E1 -31658.623,E2 -31658.623} C_VEL
LIN {X 0,Y 67.757,Z 645.663,A -85,B 0,C 180,E1 -31662.192,E2 -31662.192} C_VEL
LIN {X 0,Y 67.695,Z 646.75,A -85,B 0,C 180,E1 -31664.41,E2 -31664.41} C_VEL
LIN {X 0,Y 67.667,Z 648.242,A -85,B 0,C 180,E1 -31666.513,E2 -31666.513} C_VEL
LIN {X 0,Y 65.357,Z 660.224,A -85,B 0,C 180,E1 -31666.57,E2 -31666.57} C_VEL
LIN {X 0,Y 61.935,Z 671.835,A -85,B 0,C 180,E1 -31666.324,E2 -31666.324} C_VEL
LIN {X 0,Y 56.727,Z 684.597,A -85,B 0,C 180,E1 -31665.657,E2 -31665.657} C_VEL
LIN {X 0,Y 50.948,Z 695.536,A -85,B 0,C 180,E1 -31664.924,E2 -31664.924} C_VEL
LIN {X 0,Y 43.928,Z 706.174,A -85,B 0,C 180,E1 -31663.721,E2 -31663.721} C_VEL
LIN {X 0,Y 36.943,Z 714.888,A -85,B 0,C 180,E1 -31662.02,E2 -31662.02} C_VEL
LIN {X 0,Y 35.494,Z 716.431,A -85,B 0,C 180,E1 -31659.205,E2 -31659.205} C_VEL
LIN {X 0,Y 43.801,Z 706.169,A -85,B 0,C 180,E1 -31657.307,E2 -31657.307} C_VEL
LIN {X 0,Y 50.973,Z 695.21,A -85,B 0,C 180,E1 -31656.22,E2 -31656.22} C_VEL
LIN {X 0,Y 57.298,Z 682.979,A -85,B 0,C 180,E1 -31655.561,E2 -31655.561} C_VEL
LIN {X 0,Y 62.493,Z 669.727,A -85,B 0,C 180,E1 -31655.168,E2 -31655.168} C_VEL
LIN {X 0,Y 66.186,Z 655.988,A -85,B 0,C 180,E1 -31655.036,E2 -31655.036} C_VEL
LIN {X 0,Y 67.623,Z 648.234,A -85,B 0,C 180,E1 -31654.986,E2 -31654.986} C_VEL
LIN {X 0,Y 67.61,Z 646.92,A -85,B 0,C 180,E1 -31658.096,E2 -31658.096} C_VEL
LIN {X 0,Y 67.669,Z 646.158,A -85,B 0,C 180,E1 -31661.849,E2 -31661.849} C_VEL
LIN {X 0,Y 67.695,Z 646.75,A -85,B 0,C 180,E1 -31664.41,E2 -31664.41} C_VEL
LIN {X 0,Y 67.695,Z 646.75,A -85,B 0,C 180,E1 -31664.41,E2 -31664.41}

QRS_NEXT_CUT()

QRS_NEXT()
QRS_HOME()

END
